C03630=1077.556,71.038,-65.531,173.800,22.783,153.961
C03631=1077.550,70.789,-65.513,173.799,22.780,153.960
C03632=1077.544,70.540,-65.497,173.797,22.778,153.960
C03633=1077.539,70.291,-65.480,173.796,22.775,153.960
C03634=1077.533,70.041,-65.462,173.794,22.773,153.959
C03635=1077.527,69.791,-65.445,173.793,22.770,153.959
C03636=1077.521,69.542,-65.428,173.791,22.768,153.959
C03637=1077.516,69.293,-65.411,173.790,22.765,153.959
C03638=1077.510,69.044,-65.394,173.788,22.763,153.958
C03639=1077.504,68.794,-65.377,173.786,22.760,153.958
C03640=1077.498,68.545,-65.360,173.785,22.758,153.958
C03641=1077.492,68.295,-65.343,173.784,22.756,153.958
C03642=1077.486,68.046,-65.327,173.782,22.753,153.957
C03643=1077.481,67.797,-65.309,173.780,22.750,153.957
C03644=1077.475,67.548,-65.293,173.779,22.748,153.957
C03645=1077.469,67.298,-65.275,173.778,22.746,153.957
C03646=1077.464,67.048,-65.258,173.775,22.743,153.956
C03647=1077.457,66.799,-65.241,173.774,22.741,153.956
C03648=1077.452,66.550,-65.224,173.773,22.738,153.956
C03649=1077.446,66.300,-65.208,173.771,22.736,153.955
C03650=1077.441,66.051,-65.191,173.770,22.733,153.955
C03651=1077.435,65.802,-65.174,173.768,22.731,153.955
C03652=1077.429,65.552,-65.156,173.767,22.729,153.955
C03653=1077.423,65.303,-65.140,173.765,22.726,153.954
C03654=1077.417,65.053,-65.123,173.763,22.724,153.954
C03655=1077.411,64.804,-65.106,173.762,22.721,153.954
C03656=1077.406,64.555,-65.089,173.760,22.718,153.954
C03657=1077.400,64.305,-65.073,173.759,22.716,153.953
C03658=1077.394,64.057,-65.056,173.758,22.713,153.953
C03659=1077.389,63.807,-65.039,173.756,22.712,153.953
C03660=1077.382,63.557,-65.023,173.754,22.709,153.953
C03661=1077.376,63.277,-65.004,173.753,22.706,153.952
C03662=1077.369,62.996,-64.985,173.751,22.703,153.952
C03663=1077.362,62.715,-64.966,173.750,22.701,153.952
C03664=1077.356,62.435,-64.947,173.747,22.698,153.951
C03665=1077.349,62.185,-64.930,173.746,22.695,153.951
C03666=1077.343,61.936,-64.914,173.745,22.693,153.951
C03667=1077.338,61.686,-64.898,173.743,22.691,153.951
C03668=1077.332,61.437,-64.880,173.741,22.688,153.950
C03669=1077.326,61.188,-64.864,173.740,22.686,153.950
C03670=1077.320,60.938,-64.848,173.738,22.683,153.950
C03671=1077.314,60.689,-64.832,173.737,22.680,153.950
C03672=1077.309,60.439,-64.815,173.735,22.679,153.949
C03673=1077.303,60.191,-64.798,173.734,22.676,153.949
C03674=1077.296,59.941,-64.781,173.732,22.673,153.949
C03675=1077.291,59.691,-64.764,173.731,22.671,153.949
C03676=1077.285,59.442,-64.748,173.730,22.668,153.948
C03677=1077.279,59.192,-64.732,173.728,22.666,153.948
C03678=1077.273,58.943,-64.716,173.726,22.664,153.948
C03679=1077.268,58.694,-64.698,173.725,22.661,153.948
C03680=1077.262,58.445,-64.682,173.724,22.659,153.947
C03681=1077.256,58.195,-64.665,173.721,22.656,153.947
C03682=1077.250,57.946,-64.649,173.720,22.654,153.947
C03683=1077.244,57.696,-64.632,173.719,22.651,153.946
C03684=1077.239,57.447,-64.616,173.718,22.649,153.946
C03685=1077.233,57.198,-64.600,173.715,22.646,153.946
C03686=1077.227,56.948,-64.584,173.714,22.644,153.946
C03687=1077.221,56.699,-64.567,173.713,22.642,153.945
C03688=1077.215,56.450,-64.550,173.712,22.639,153.945
C03689=1077.209,56.200,-64.534,173.710,22.636,153.945
C03690=1077.203,55.951,-64.517,173.708,22.634,153.945
C03691=1077.197,55.702,-64.501,173.707,22.631,153.944
C03692=1077.191,55.452,-64.485,173.706,22.629,153.944
C03693=1077.186,55.203,-64.468,173.704,22.626,153.944
C03694=1077.180,54.953,-64.452,173.702,22.624,153.944
C03695=1077.174,54.704,-64.435,173.701,22.622,153.943
C03696=1077.168,54.455,-64.419,173.700,22.619,153.943
C03697=1077.162,54.205,-64.403,173.698,22.617,153.943
C03698=1077.157,53.956,-64.386,173.696,22.614,153.942
C03699=1077.151,53.706,-64.370,173.695,22.612,153.942
C03700=1077.145,53.457,-64.354,173.694,22.609,153.942
C03701=1077.139,53.208,-64.337,173.692,22.606,153.942
C03702=1077.133,52.958,-64.321,173.691,22.604,153.941
C03703=1077.128,52.709,-64.304,173.689,22.602,153.941
C03704=1077.122,52.459,-64.288,173.688,22.599,153.941
C03705=1077.116,52.210,-64.272,173.686,22.596,153.940
C03706=1077.110,51.961,-64.255,173.685,22.594,153.940
C03707=1077.105,51.711,-64.240,173.683,22.592,153.940
C03708=1077.099,51.461,-64.224,173.681,22.589,153.940
C03709=1077.093,51.212,-64.207,173.680,22.587,153.939
C03710=1077.087,50.962,-64.190,173.679,22.584,153.939
C03711=1077.082,50.713,-64.174,173.678,22.582,153.939
C03712=1077.076,50.464,-64.158,173.675,22.579,153.939
C03713=1077.070,50.215,-64.142,173.674,22.577,153.938
C03714=1077.064,49.966,-64.126,173.673,22.574,153.938
C03715=1077.059,49.716,-64.110,173.672,22.572,153.938
C03716=1077.053,49.466,-64.093,173.670,22.569,153.937
C03717=1077.047,49.217,-64.077,173.668,22.566,153.937
C03718=1077.042,48.967,-64.061,173.667,22.564,153.937
C03719=1077.036,48.718,-64.045,173.666,22.562,153.937
C03720=1077.030,48.469,-64.028,173.665,22.559,153.936
C03721=1077.024,48.219,-64.013,173.663,22.556,153.936
C03722=1077.019,47.970,-63.997,173.661,22.554,153.936
C03723=1077.013,47.721,-63.981,173.660,22.551,153.935
C03724=1077.007,47.471,-63.964,173.659,22.549,153.935
C03725=1077.000,47.189,-63.946,173.657,22.546,153.935
C03726=1076.994,46.909,-63.928,173.655,22.543,153.935
C03727=1076.988,46.628,-63.909,173.654,22.540,153.934
C03728=1076.982,46.347,-63.892,173.651,22.538,153.934
C03729=1076.976,46.097,-63.875,173.650,22.535,153.934
C03730=1076.970,45.848,-63.859,173.649,22.533,153.933
C03731=1076.964,45.599,-63.843,173.648,22.530,153.933
C03732=1076.959,45.349,-63.828,173.646,22.527,153.933
C03733=1076.953,45.100,-63.812,173.644,22.525,153.932
C03734=1076.947,44.851,-63.795,173.643,22.523,153.932
C03735=1076.941,44.601,-63.780,173.642,22.520,153.932
C03736=1076.936,44.351,-63.763,173.641,22.518,153.932
C03737=1076.930,44.103,-63.748,173.639,22.515,153.931
C03738=1076.925,43.853,-63.732,173.637,22.512,153.931
C03739=1076.919,43.603,-63.716,173.636,22.510,153.931
C03740=1076.913,43.354,-63.700,173.635,22.508,153.930
C03741=1076.907,43.104,-63.684,173.633,22.505,153.930
C03742=1076.901,42.855,-63.668,173.632,22.502,153.930
C03743=1076.896,42.606,-63.652,173.630,22.500,153.930
C03744=1076.890,42.356,-63.636,173.629,22.497,153.929
C03745=1076.884,42.107,-63.620,173.627,22.494,153.929
C03746=1076.878,41.857,-63.605,173.626,22.492,153.929
C03747=1076.872,41.608,-63.589,173.625,22.490,153.928
C03748=1076.866,41.359,-63.573,173.623,22.488,153.928
C03749=1076.861,41.109,-63.557,173.621,22.485,153.928
C03750=1076.855,40.860,-63.541,173.620,22.482,153.928
C03751=1076.849,40.610,-63.526,173.619,22.480,153.927
C03752=1076.843,40.360,-63.509,173.617,22.478,153.927
C03753=1076.838,40.111,-63.494,173.616,22.475,153.927
C03754=1076.831,39.862,-63.479,173.614,22.472,153.927
C03755=1076.826,39.613,-63.462,173.613,22.470,153.926
C03756=1076.820,39.363,-63.447,173.612,22.467,153.926
C03757=1076.814,39.113,-63.430,173.610,22.465,153.926
C03758=1076.809,38.864,-63.415,173.608,22.462,153.925
C03759=1076.803,38.615,-63.399,173.607,22.460,153.925
C03760=1076.797,38.365,-63.383,173.606,22.457,153.925
C03761=1076.791,38.116,-63.368,173.605,22.455,153.925
C03762=1076.786,37.867,-63.353,173.603,22.452,153.924
C03763=1076.780,37.617,-63.337,173.601,22.449,153.924
C03764=1076.774,37.367,-63.321,173.600,22.448,153.924
C03765=1076.768,37.118,-63.306,173.599,22.445,153.924
C03766=1076.762,36.869,-63.290,173.597,22.443,153.923
C03767=1076.757,36.619,-63.274,173.595,22.440,153.923
C03768=1076.750,36.370,-63.259,173.594,22.437,153.923
C03769=1076.744,36.120,-63.243,173.593,22.435,153.922
C03770=1076.738,35.871,-63.227,173.592,22.433,153.922
C03771=1076.732,35.622,-63.212,173.590,22.430,153.922
C03772=1076.727,35.372,-63.197,173.588,22.427,153.922
C03773=1076.721,35.122,-63.181,173.587,22.425,153.921
C03774=1076.715,34.873,-63.166,173.586,22.423,153.921
C03775=1076.709,34.624,-63.150,173.584,22.420,153.921
C03776=1076.704,34.374,-63.134,173.582,22.418,153.921
C03777=1076.697,34.124,-63.119,173.581,22.415,153.920
C03778=1076.691,33.875,-63.103,173.580,22.413,153.920
C03779=1076.686,33.626,-63.088,173.579,22.410,153.920
C03780=1076.680,33.376,-63.073,173.577,22.408,153.919
C03781=1076.674,33.127,-63.057,173.575,22.405,153.919
C03782=1076.669,32.878,-63.042,173.574,22.403,153.919
C03783=1076.662,32.628,-63.027,173.573,22.400,153.919
C03784=1076.656,32.379,-63.010,173.571,22.398,153.918
C03785=1076.651,32.130,-62.996,173.570,22.396,153.918
C03786=1076.645,31.880,-62.980,173.568,22.393,153.918
C03787=1076.639,31.630,-62.965,173.567,22.390,153.918
C03788=1076.633,31.381,-62.949,173.566,22.388,153.917
C03789=1076.626,31.100,-62.932,173.564,22.385,153.917
C03790=1076.620,30.819,-62.914,173.563,22.382,153.917
C03791=1076.614,30.538,-62.897,173.560,22.379,153.916
C03792=1076.607,30.256,-62.880,173.559,22.377,153.916
C03793=1076.602,30.007,-62.865,173.558,22.374,153.916
C03794=1076.595,29.757,-62.850,173.557,22.372,153.916
C03795=1076.590,29.509,-62.834,173.555,22.369,153.915
C03796=1076.584,29.259,-62.819,173.553,22.367,153.915
C03797=1076.578,29.009,-62.803,173.552,22.364,153.915
C03798=1076.573,28.760,-62.788,173.551,22.362,153.914
C03799=1076.567,28.510,-62.773,173.550,22.359,153.914
C03800=1076.561,28.261,-62.757,173.548,22.356,153.914
C03801=1076.555,28.012,-62.742,173.546,22.354,153.914
C03802=1076.548,27.762,-62.727,173.545,22.352,153.913
C03803=1076.543,27.512,-62.712,173.544,22.350,153.913
C03804=1076.537,27.263,-62.697,173.543,22.347,153.913
C03805=1076.531,27.013,-62.682,173.541,22.344,153.913
C03806=1076.525,26.764,-62.666,173.539,22.342,153.912
C03807=1076.520,26.515,-62.651,173.538,22.339,153.912
C03808=1076.513,26.265,-62.636,173.537,22.337,153.912
C03809=1076.508,26.015,-62.620,173.536,22.335,153.911
C03810=1076.502,25.767,-62.606,173.533,22.332,153.911
C03811=1076.495,25.517,-62.591,173.532,22.330,153.911
C03812=1076.490,25.268,-62.576,173.531,22.327,153.911
C03813=1076.484,25.018,-62.561,173.530,22.325,153.910
C03814=1076.478,24.768,-62.545,173.528,22.322,153.910
C03815=1076.473,24.519,-62.531,173.526,22.320,153.910
C03816=1076.467,24.269,-62.515,173.525,22.317,153.910
C03817=1076.461,24.019,-62.500,173.524,22.315,153.909
C03818=1076.455,23.770,-62.486,173.523,22.313,153.909
C03819=1076.449,23.520,-62.470,173.521,22.310,153.909
C03820=1076.443,23.271,-62.455,173.519,22.307,153.909
C03821=1076.437,23.022,-62.441,173.518,22.305,153.908
C03822=1076.431,22.772,-62.425,173.517,22.303,153.908
C03823=1076.426,22.523,-62.410,173.516,22.300,153.908
C03824=1076.420,22.273,-62.395,173.514,22.298,153.907
C03825=1076.414,22.024,-62.380,173.512,22.295,153.907
C03826=1076.408,21.774,-62.365,173.511,22.293,153.907
C03827=1076.403,21.525,-62.350,173.510,22.290,153.907
C03828=1076.396,21.275,-62.335,173.508,22.288,153.906
C03829=1076.391,21.026,-62.321,173.507,22.286,153.906
C03830=1076.385,20.776,-62.305,173.505,22.283,153.906
C03831=1076.379,20.527,-62.290,173.504,22.280,153.906
C03832=1076.373,20.278,-62.275,173.503,22.278,153.905
C03833=1076.367,20.028,-62.260,173.502,22.275,153.905
C03834=1076.361,19.779,-62.245,173.500,22.273,153.905
C03835=1076.355,19.529,-62.231,173.498,22.271,153.905
C03836=1076.350,19.280,-62.215,173.497,22.268,153.904
C03837=1076.344,19.030,-62.200,173.496,22.266,153.904
C03838=1076.338,18.781,-62.187,173.494,22.263,153.904
C03839=1076.332,18.531,-62.172,173.493,22.261,153.903
C03840=1076.327,18.282,-62.156,173.491,22.258,153.903
C03841=1076.320,18.032,-62.141,173.490,22.256,153.903
C03842=1076.314,17.783,-62.127,173.488,22.254,153.903
C03843=1076.308,17.534,-62.112,173.487,22.251,153.902
C03844=1076.302,17.284,-62.096,173.486,22.249,153.902
C03845=1076.297,17.034,-62.083,173.485,22.246,153.902
C03846=1076.291,16.784,-62.068,173.483,22.243,153.902
C03847=1076.285,16.535,-62.053,173.482,22.241,153.901
C03848=1076.278,16.286,-62.038,173.480,22.239,153.901
C03849=1076.273,16.037,-62.023,173.479,22.236,153.901
C03850=1076.267,15.786,-62.009,173.478,22.234,153.900
C03851=1076.262,15.537,-61.994,173.476,22.231,153.900
C03852=1076.255,15.288,-61.979,173.474,22.229,153.900
C03853=1076.250,15.008,-61.963,173.473,22.226,153.900
C03854=1076.243,14.729,-61.946,173.471,22.223,153.899
C03855=1076.236,14.449,-61.930,173.470,22.220,153.899
C03856=1076.230,14.170,-61.914,173.468,22.218,153.899
C03857=1076.223,13.920,-61.899,173.467,22.216,153.899
C03858=1076.217,13.671,-61.884,173.465,22.213,153.898
C03859=1076.211,13.421,-61.870,173.464,22.211,153.898
C03860=1076.206,13.172,-61.856,173.463,22.208,153.898
C03861=1076.199,12.922,-61.841,173.462,22.206,153.898
C03862=1076.193,12.673,-61.826,173.460,22.203,153.897
C03863=1076.187,12.423,-61.812,173.458,22.201,153.897
C03864=1076.182,12.174,-61.797,173.457,22.199,153.897
C03865=1076.175,11.924,-61.782,173.456,22.196,153.896
C03866=1076.170,11.675,-61.768,173.455,22.194,153.896
C03867=1076.163,11.425,-61.753,173.453,22.192,153.896
C03868=1076.158,11.176,-61.739,173.451,22.189,153.896
C03869=1076.151,10.926,-61.725,173.450,22.186,153.895
C03870=1076.146,10.677,-61.710,173.449,22.184,153.895
C03871=1076.140,10.427,-61.696,173.447,22.182,153.895
C03872=1076.134,10.178,-61.681,173.446,22.180,153.895
C03873=1076.127,9.928,-61.666,173.444,22.177,153.894
C03874=1076.122,9.678,-61.652,173.443,22.175,153.894
C03875=1076.116,9.429,-61.637,173.442,22.172,153.894
C03876=1076.110,9.179,-61.624,173.440,22.170,153.894
C03877=1076.104,8.930,-61.609,173.439,22.167,153.893
C03878=1076.098,8.681,-61.594,173.438,22.165,153.893
C03879=1076.092,8.431,-61.580,173.436,22.163,153.893
C03880=1076.086,8.181,-61.565,173.434,22.160,153.893
C03881=1076.081,7.932,-61.551,173.433,22.158,153.892
C03882=1076.074,7.682,-61.536,173.432,22.155,153.892
C03883=1076.069,7.432,-61.523,173.431,22.153,153.892
C03884=1076.063,7.184,-61.508,173.429,22.151,153.892
C03885=1076.057,6.933,-61.494,173.427,22.148,153.891
C03886=1076.051,6.684,-61.479,173.426,22.146,153.891
C03887=1076.045,6.434,-61.465,173.425,22.143,153.891
C03888=1076.039,6.185,-61.450,173.424,22.141,153.891
C03889=1076.034,5.935,-61.437,173.422,22.139,153.890
C03890=1076.027,5.686,-61.422,173.421,22.136,153.890
C03891=1076.022,5.436,-61.408,173.419,22.133,153.890
C03892=1076.016,5.187,-61.393,173.418,22.131,153.890
C03893=1076.009,4.937,-61.379,173.416,22.129,153.889
C03894=1076.004,4.688,-61.365,173.415,22.127,153.889
C03895=1075.998,4.439,-61.351,173.414,22.124,153.889
C03896=1075.992,4.189,-61.337,173.412,22.121,153.889
C03897=1075.986,3.940,-61.322,173.411,22.119,153.888
C03898=1075.980,3.689,-61.308,173.409,22.117,153.888
C03899=1075.974,3.440,-61.293,173.408,22.114,153.888
C03900=1075.969,3.191,-61.280,173.407,22.112,153.887
C03901=1075.963,2.941,-61.266,173.406,22.109,153.887
C03902=1075.957,2.692,-61.251,173.403,22.107,153.887
C03903=1075.952,2.442,-61.237,173.402,22.105,153.887
C03904=1075.945,2.193,-61.223,173.401,22.102,153.887
C03905=1075.939,1.943,-61.209,173.400,22.100,153.886
C03906=1075.933,1.693,-61.195,173.399,22.098,153.886
C03907=1075.928,1.444,-61.180,173.397,22.095,153.886
C03908=1075.922,1.194,-61.166,173.395,22.092,153.886
C03909=1075.916,0.945,-61.152,173.394,22.090,153.885
C03910=1075.910,0.696,-61.138,173.393,22.088,153.885
C03911=1075.905,0.446,-61.124,173.391,22.086,153.885
C03912=1075.899,0.196,-61.109,173.390,22.083,153.884
C03913=1075.893,-0.053,-61.096,173.389,22.081,153.884
C03914=1075.887,-0.302,-61.082,173.387,22.078,153.884
C03915=1075.881,-0.553,-61.067,173.386,22.075,153.884
C03916=1075.875,-0.802,-61.054,173.384,22.073,153.883
C03917=1075.869,-1.080,-61.038,173.383,22.071,153.883
C03918=1075.862,-1.357,-61.023,173.381,22.068,153.883
C03919=1075.857,-1.635,-61.006,173.380,22.065,153.883
C03920=1075.849,-1.913,-60.991,173.379,22.063,153.882
C03921=1075.844,-2.162,-60.977,173.377,22.060,153.882
C03922=1075.837,-2.411,-60.963,173.375,22.058,153.882
C03923=1075.832,-2.661,-60.949,173.374,22.055,153.882
C03924=1075.826,-2.910,-60.935,173.373,22.053,153.881
C03925=1075.820,-3.161,-60.921,173.372,22.050,153.881
C03926=1075.815,-3.410,-60.907,173.370,22.048,153.881
C03927=1075.808,-3.659,-60.893,173.368,22.046,153.881
C03928=1075.803,-3.908,-60.879,173.367,22.043,153.880
C03929=1075.796,-4.158,-60.865,173.366,22.041,153.880
C03930=1075.791,-4.408,-60.852,173.365,22.039,153.880
C03931=1075.785,-4.657,-60.838,173.363,22.036,153.880
C03932=1075.778,-4.907,-60.823,173.362,22.034,153.879
C03933=1075.773,-5.156,-60.810,173.360,22.031,153.879
C03934=1075.767,-5.406,-60.796,173.359,22.030,153.879
C03935=1075.761,-5.655,-60.782,173.357,22.027,153.879
C03936=1075.755,-5.905,-60.768,173.356,22.025,153.878
C03937=1075.749,-6.155,-60.755,173.355,22.023,153.878
C03938=1075.743,-6.404,-60.741,173.354,22.020,153.878
C03939=1075.737,-6.654,-60.728,173.352,22.018,153.878
C03940=1075.731,-6.904,-60.714,173.350,22.015,153.878
C03941=1075.725,-7.153,-60.699,173.349,22.013,153.877
C03942=1075.719,-7.402,-60.686,173.348,22.010,153.877
C03943=1075.713,-7.652,-60.672,173.346,22.009,153.877
C03944=1075.707,-7.901,-60.659,173.345,22.006,153.876
C03945=1075.701,-8.151,-60.644,173.344,22.004,153.876
C03946=1075.696,-8.401,-60.630,173.342,22.001,153.876
C03947=1075.689,-8.650,-60.617,173.341,21.999,153.876
C03948=1075.684,-8.900,-60.603,173.339,21.997,153.876
C03949=1075.678,-9.149,-60.590,173.338,21.994,153.875
C03950=1075.672,-9.399,-60.576,173.337,21.992,153.875
C03951=1075.665,-9.648,-60.563,173.335,21.990,153.875
C03952=1075.660,-9.898,-60.549,173.334,21.988,153.875
C03953=1075.654,-10.147,-60.535,173.332,21.985,153.874
C03954=1075.648,-10.397,-60.522,173.331,21.983,153.874
C03955=1075.641,-10.647,-60.508,173.330,21.980,153.874
C03956=1075.636,-10.896,-60.494,173.328,21.978,153.874
C03957=1075.630,-11.146,-60.480,173.327,21.976,153.873
C03958=1075.624,-11.395,-60.467,173.326,21.973,153.873
C03959=1075.619,-11.645,-60.453,173.323,21.971,153.873
C03960=1075.613,-11.894,-60.440,173.322,21.969,153.873
C03961=1075.607,-12.144,-60.426,173.321,21.966,153.872
C03962=1075.600,-12.394,-60.412,173.320,21.964,153.872
C03963=1075.595,-12.644,-60.399,173.319,21.962,153.872
C03964=1075.589,-12.893,-60.386,173.317,21.959,153.872
C03965=1075.583,-13.143,-60.372,173.316,21.957,153.872
C03966=1075.577,-13.392,-60.359,173.314,21.954,153.871
C03967=1075.572,-13.641,-60.345,173.313,21.952,153.871
C03968=1075.565,-13.891,-60.332,173.311,21.950,153.871
C03969=1075.560,-14.140,-60.318,173.310,21.948,153.871
C03970=1075.554,-14.390,-60.304,173.309,21.946,153.870
C03971=1075.548,-14.640,-60.291,173.308,21.943,153.870
C03972=1075.542,-14.890,-60.278,173.306,21.941,153.870
C03973=1075.536,-15.139,-60.264,173.304,21.938,153.870
C03974=1075.530,-15.389,-60.251,173.303,21.936,153.869
C03975=1075.524,-15.638,-60.237,173.302,21.934,153.869
C03976=1075.518,-15.887,-60.223,173.300,21.931,153.869
C03977=1075.513,-16.137,-60.211,173.299,21.930,153.869
C03978=1075.506,-16.387,-60.198,173.298,21.927,153.869
C03979=1075.500,-16.637,-60.183,173.296,21.925,153.868
C03980=1075.494,-16.886,-60.170,173.294,21.922,153.868
C03981=1075.488,-17.162,-60.156,173.293,21.920,153.868
C03982=1075.481,-17.437,-60.141,173.292,21.918,153.868
C03983=1075.474,-17.714,-60.126,173.290,21.915,153.867
C03984=1075.468,-17.990,-60.112,173.289,21.912,153.867
C03985=1075.462,-18.240,-60.098,173.287,21.911,153.867
C03986=1075.456,-18.489,-60.085,173.286,21.908,153.867
C03987=1075.450,-18.738,-60.071,173.284,21.906,153.867
C03988=1075.444,-18.988,-60.059,173.283,21.903,153.866
C03989=1075.438,-19.237,-60.045,173.281,21.901,153.866
C03990=1075.432,-19.487,-60.032,173.280,21.899,153.866
C03991=1075.426,-19.736,-60.018,173.279,21.897,153.866
C03992=1075.420,-19.986,-60.006,173.277,21.894,153.865
C03993=1075.413,-20.236,-59.992,173.276,21.892,153.865
C03994=1075.408,-20.486,-59.978,173.275,21.890,153.865
C03995=1075.402,-20.736,-59.966,173.273,21.888,153.865
C03996=1075.396,-20.985,-59.952,173.271,21.885,153.865
C03997=1075.390,-21.234,-59.939,173.270,21.883,153.864
C03998=1075.384,-21.484,-59.926,173.269,21.881,153.864
C03999=1075.378,-21.734,-59.913,173.267,21.879,153.864
C04000=1075.372,-21.983,-59.900,173.266,21.876,153.864
C04001=1075.367,-22.233,-59.886,173.265,21.874,153.863
C04002=1075.361,-22.482,-59.873,173.263,21.872,153.863
C04003=1075.355,-22.732,-59.861,173.261,21.870,153.863
C04004=1075.348,-22.981,-59.847,173.260,21.867,153.863
C04005=1075.343,-23.231,-59.833,173.259,21.865,153.863
C04006=1075.337,-23.481,-59.821,173.258,21.863,153.862
C04007=1075.331,-23.730,-59.808,173.256,21.861,153.862
C04008=1075.325,-23.980,-59.795,173.255,21.858,153.862
C04009=1075.319,-24.229,-59.782,173.253,21.856,153.862
C04010=1075.313,-24.479,-59.768,173.252,21.853,153.861
C04011=1075.307,-24.729,-59.755,173.250,21.852,153.861
C04012=1075.301,-24.978,-59.742,173.249,21.849,153.861
C04013=1075.295,-25.228,-59.730,173.248,21.847,153.861
C04014=1075.290,-25.478,-59.716,173.246,21.845,153.861
C04015=1075.284,-25.727,-59.703,173.245,21.843,153.860
C04016=1075.278,-25.977,-59.690,173.244,21.841,153.860
C04017=1075.272,-26.227,-59.677,173.242,21.838,153.860
C04018=1075.266,-26.475,-59.664,173.240,21.836,153.860
C04019=1075.261,-26.725,-59.651,173.239,21.833,153.860
C04020=1075.255,-26.975,-59.638,173.238,21.832,153.859
C04021=1075.249,-27.224,-59.625,173.237,21.829,153.859
C04022=1075.243,-27.474,-59.612,173.235,21.827,153.859
C04023=1075.237,-27.724,-59.600,173.234,21.825,153.859
C04024=1075.230,-27.973,-59.586,173.232,21.822,153.859
C04025=1075.225,-28.223,-59.574,173.230,21.820,153.858
C04026=1075.218,-28.472,-59.560,173.229,21.818,153.858
C04027=1075.212,-28.722,-59.548,173.228,21.816,153.858
C04028=1075.207,-28.972,-59.535,173.227,21.814,153.858
C04029=1075.200,-29.221,-59.522,173.225,21.812,153.858
C04030=1075.194,-29.471,-59.510,173.224,21.810,153.857
C04031=1075.188,-29.720,-59.496,173.223,21.808,153.857
C04032=1075.182,-29.970,-59.484,173.220,21.805,153.857
C04033=1075.176,-30.220,-59.471,173.219,21.803,153.857
C04034=1075.170,-30.469,-59.458,173.218,21.801,153.857
C04035=1075.164,-30.719,-59.445,173.216,21.799,153.856
C04036=1075.158,-30.968,-59.432,173.215,21.796,153.856
C04037=1075.152,-31.218,-59.420,173.214,21.795,153.856
C04038=1075.146,-31.468,-59.407,173.212,21.793,153.856
C04039=1075.140,-31.717,-59.394,173.211,21.790,153.856
C04040=1075.134,-31.967,-59.381,173.209,21.788,153.855
C04041=1075.129,-32.216,-59.369,173.208,21.786,153.855
C04042=1075.123,-32.466,-59.356,173.207,21.783,153.855
C04043=1075.117,-32.716,-59.343,173.205,21.781,153.855
C04044=1075.111,-32.966,-59.331,173.204,21.779,153.855
C04045=1075.104,-33.240,-59.316,173.203,21.777,153.854
C04046=1075.097,-33.516,-59.303,173.200,21.775,153.854
C04047=1075.091,-33.791,-59.289,173.199,21.772,153.854
C04048=1075.084,-34.066,-59.274,173.198,21.770,153.854
C04049=1075.078,-34.316,-59.262,173.197,21.768,153.854
C04050=1075.072,-34.566,-59.249,173.194,21.765,153.853
C04051=1075.066,-34.814,-59.236,173.193,21.763,153.853
C04052=1075.061,-35.064,-59.224,173.192,21.761,153.853
C04053=1075.055,-35.314,-59.211,173.190,21.759,153.853
C04054=1075.049,-35.564,-59.199,173.189,21.757,153.853
C04055=1075.043,-35.814,-59.186,173.188,21.755,153.852
C04056=1075.037,-36.063,-59.173,173.187,21.753,153.852
C04057=1075.031,-36.313,-59.160,173.185,21.751,153.852
C04058=1075.025,-36.562,-59.149,173.183,21.748,153.852
C04059=1075.019,-36.812,-59.136,173.182,21.746,153.852
C04060=1075.013,-37.062,-59.124,173.180,21.744,153.852
C04061=1075.007,-37.311,-59.110,173.179,21.742,153.851
C04062=1075.001,-37.561,-59.098,173.178,21.740,153.851
C04063=1074.995,-37.810,-59.086,173.176,21.738,153.851
C04064=1074.989,-38.060,-59.073,173.175,21.736,153.851
C04065=1074.984,-38.310,-59.060,173.174,21.734,153.851
C04066=1074.978,-38.560,-59.048,173.173,21.731,153.850
C04067=1074.971,-38.809,-59.035,173.170,21.729,153.850
C04068=1074.965,-39.058,-59.023,173.169,21.727,153.850
C04069=1074.959,-39.308,-59.011,173.168,21.725,153.850
C04070=1074.954,-39.557,-58.998,173.166,21.723,153.850
C04071=1074.947,-39.807,-58.986,173.165,21.721,153.850
C04072=1074.941,-40.057,-58.973,173.164,21.719,153.849
C04073=1074.935,-40.307,-58.961,173.162,21.717,153.849
C04074=1074.929,-40.557,-58.948,173.161,21.715,153.849
C04075=1074.923,-40.806,-58.937,173.159,21.713,153.849
C04076=1074.917,-41.055,-58.923,173.157,21.710,153.849
C04077=1074.911,-41.305,-58.911,173.156,21.708,153.849
C04078=1074.905,-41.555,-58.898,173.154,21.707,153.848
C04079=1074.898,-41.804,-58.886,173.153,21.704,153.848
C04080=1074.893,-42.053,-58.874,173.152,21.702,153.848
C04081=1074.887,-42.303,-58.862,173.151,21.700,153.848
C04082=1074.881,-42.553,-58.850,173.149,21.698,153.848
C04083=1074.875,-42.803,-58.837,173.148,21.696,153.848
C04084=1074.869,-43.053,-58.825,173.146,21.694,153.847
C04085=1074.863,-43.301,-58.813,173.144,21.692,153.847
C04086=1074.857,-43.551,-58.800,173.143,21.690,153.847
C04087=1074.851,-43.801,-58.788,173.142,21.688,153.847
C04088=1074.844,-44.051,-58.776,173.140,21.686,153.847
C04089=1074.839,-44.300,-58.764,173.139,21.684,153.846
C04090=1074.833,-44.550,-58.751,173.138,21.682,153.846
C04091=1074.827,-44.800,-58.739,173.136,21.680,153.846
C04092=1074.821,-45.049,-58.727,173.135,21.678,153.846
C04093=1074.815,-45.298,-58.715,173.133,21.676,153.846
C04094=1074.809,-45.548,-58.702,173.132,21.674,153.846
C04095=1074.803,-45.798,-58.690,173.130,21.672,153.846
C04096=1074.797,-46.048,-58.678,173.129,21.669,153.845
C04097=1074.791,-46.297,-58.667,173.127,21.667,153.845
C04098=1074.785,-46.547,-58.654,173.126,21.665,153.845
C04099=1074.779,-46.797,-58.641,173.125,21.663,153.845
C04100=1074.773,-47.046,-58.630,173.123,21.661,153.845
C04101=1074.767,-47.296,-58.617,173.122,21.659,153.845
C04102=1074.761,-47.546,-58.605,173.120,21.657,153.844
C04103=1074.755,-47.795,-58.593,173.119,21.656,153.844
C04104=1074.749,-48.044,-58.581,173.118,21.654,153.844
C04105=1074.743,-48.294,-58.568,173.116,21.651,153.844
C04106=1074.737,-48.545,-58.557,173.114,21.649,153.844
C04107=1074.732,-48.794,-58.545,173.113,21.647,153.844
C04108=1074.726,-49.044,-58.532,173.111,21.645,153.843
C04109=1074.719,-49.319,-58.519,173.110,21.643,153.843
C04110=1074.713,-49.595,-58.506,173.109,21.641,153.843
C04111=1074.706,-49.870,-58.492,173.107,21.639,153.843
C04112=1074.699,-50.146,-58.479,173.105,21.637,153.843
C04113=1074.694,-50.395,-58.467,173.104,21.634,153.842
C04114=1074.688,-50.645,-58.455,173.103,21.633,153.842
C04115=1074.681,-50.895,-58.443,173.101,21.631,153.842
C04116=1074.675,-51.144,-58.431,173.100,21.629,153.842
C04117=1074.669,-51.393,-58.419,173.098,21.626,153.842
C04118=1074.663,-51.644,-58.408,173.096,21.625,153.842
C04119=1074.657,-51.893,-58.395,173.095,21.623,153.842
C04120=1074.650,-52.143,-58.383,173.093,21.621,153.842
C04121=1074.644,-52.392,-58.372,173.092,21.619,153.841
C04122=1074.638,-52.642,-58.360,173.091,21.617,153.841
C04123=1074.632,-52.892,-58.348,173.089,21.615,153.841
C04124=1074.626,-53.141,-58.336,173.088,21.613,153.841
C04125=1074.620,-53.391,-58.324,173.086,21.611,153.841
C04126=1074.613,-53.641,-58.313,173.085,21.610,153.841
C04127=1074.607,-53.890,-58.301,173.084,21.608,153.841
C04128=1074.601,-54.140,-58.288,173.082,21.606,153.840
C04129=1074.595,-54.390,-58.277,173.080,21.604,153.840
C04130=1074.589,-54.639,-58.266,173.079,21.602,153.840
C04131=1074.583,-54.889,-58.253,173.077,21.600,153.840
C04132=1074.577,-55.139,-58.242,173.076,21.598,153.840
C04133=1074.571,-55.388,-58.230,173.074,21.596,153.840
C04134=1074.565,-55.638,-58.218,173.073,21.594,153.840
C04135=1074.559,-55.888,-58.206,173.072,21.593,153.840
C04136=1074.553,-56.137,-58.195,173.070,21.591,153.840
C04137=1074.547,-56.386,-58.182,173.069,21.589,153.839
C04138=1074.540,-56.637,-58.171,173.067,21.587,153.839
C04139=1074.534,-56.886,-58.159,173.066,21.585,153.839
C04140=1074.529,-57.136,-58.148,173.065,21.583,153.839
C04141=1074.522,-57.386,-58.136,173.062,21.581,153.839
C04142=1074.516,-57.634,-58.124,173.061,21.579,153.839
C04143=1074.510,-57.885,-58.113,173.060,21.577,153.839
C04144=1074.504,-58.134,-58.101,173.058,21.575,153.838
C04145=1074.498,-58.384,-58.089,173.057,21.573,153.838
C04146=1074.491,-58.634,-58.077,173.055,21.572,153.838
C04147=1074.486,-58.883,-58.066,173.054,21.570,153.838
C04148=1074.480,-59.133,-58.054,173.053,21.568,153.838
C04149=1074.474,-59.382,-58.042,173.051,21.566,153.838
C04150=1074.467,-59.632,-58.031,173.050,21.564,153.838
C04151=1074.461,-59.882,-58.019,173.048,21.563,153.838
C04152=1074.456,-60.131,-58.008,173.047,21.561,153.837
C04153=1074.449,-60.381,-57.996,173.046,21.559,153.837
C04154=1074.444,-60.631,-57.984,173.044,21.557,153.837
C04155=1074.437,-60.880,-57.972,173.042,21.555,153.837
C04156=1074.432,-61.130,-57.961,173.040,21.553,153.837
C04157=1074.425,-61.379,-57.949,173.039,21.551,153.837
C04158=1074.419,-61.630,-57.938,173.038,21.549,153.837
C04159=1074.413,-61.879,-57.926,173.036,21.548,153.837
C04160=1074.407,-62.129,-57.915,173.035,21.546,153.837
C04161=1074.401,-62.378,-57.903,173.033,21.544,153.836
C04162=1074.395,-62.628,-57.892,173.032,21.542,153.836
C04163=1074.390,-62.878,-57.880,173.030,21.541,153.836
C04164=1074.383,-63.127,-57.868,173.029,21.539,153.836
C04165=1074.377,-63.377,-57.858,173.028,21.537,153.836
C04166=1074.371,-63.626,-57.846,173.026,21.535,153.836
C04167=1074.366,-63.876,-57.834,173.025,21.533,153.836
C04168=1074.359,-64.126,-57.822,173.023,21.531,153.836
C04169=1074.353,-64.375,-57.811,173.022,21.529,153.835
C04170=1074.347,-64.626,-57.800,173.020,21.528,153.835
C04171=1074.341,-64.874,-57.788,173.018,21.526,153.835
C04172=1074.335,-65.125,-57.777,173.017,21.524,153.835
C04173=1074.329,-65.402,-57.765,173.016,21.522,153.835
C04174=1074.322,-65.678,-57.751,173.014,21.520,153.835
C04175=1074.315,-65.956,-57.739,173.012,21.518,153.835
C04176=1074.308,-66.232,-57.726,173.010,21.516,153.835
C04177=1074.302,-66.482,-57.715,173.009,21.514,153.835
C04178=1074.297,-66.731,-57.704,173.008,21.512,153.834
C04179=1074.290,-66.981,-57.692,173.006,21.511,153.834
C04180=1074.285,-67.231,-57.680,173.005,21.509,153.834
C04181=1074.279,-67.481,-57.669,173.003,21.507,153.834
C04182=1074.273,-67.730,-57.658,173.002,21.505,153.834
C04183=1074.266,-67.980,-57.646,173.000,21.503,153.834
C04184=1074.261,-68.229,-57.635,172.999,21.502,153.834
C04185=1074.255,-68.480,-57.624,172.998,21.500,153.834
C04186=1074.249,-68.729,-57.612,172.996,21.498,153.834
C04187=1074.243,-68.978,-57.601,172.995,21.496,153.833
C04188=1074.237,-69.228,-57.590,172.993,21.495,153.833
C04189=1074.231,-69.478,-57.579,172.991,21.492,153.833
C04190=1074.224,-69.727,-57.567,172.990,21.490,153.833
C04191=1074.219,-69.977,-57.556,172.988,21.489,153.833
C04192=1074.214,-70.227,-57.545,172.987,21.487,153.833
C04193=1074.207,-70.477,-57.534,172.985,21.486,153.833
C04194=1074.201,-70.726,-57.522,172.984,21.484,153.833
C04195=1074.195,-70.976,-57.511,172.982,21.482,153.833
C04196=1074.189,-71.225,-57.500,172.981,21.480,153.833
C04197=1074.183,-71.475,-57.489,172.980,21.478,153.832
C04198=1074.177,-71.725,-57.478,172.978,21.477,153.832
C04199=1074.172,-71.974,-57.465,172.977,21.475,153.832
C04200=1074.166,-72.224,-57.455,172.975,21.473,153.832
C04201=1074.160,-72.474,-57.443,172.974,21.472,153.832
C04202=1074.154,-72.723,-57.432,172.972,21.470,153.832
C04203=1074.148,-72.973,-57.422,172.971,21.468,153.832
C04204=1074.142,-73.223,-57.410,172.969,21.466,153.832
C04205=1074.136,-73.472,-57.399,172.968,21.464,153.832
C04206=1074.130,-73.722,-57.388,172.966,21.463,153.832
C04207=1074.125,-73.972,-57.376,172.965,21.461,153.831
C04208=1074.118,-74.221,-57.366,172.964,21.460,153.831
C04209=1074.112,-74.471,-57.355,172.962,21.458,153.831
C04210=1074.106,-74.721,-57.344,172.961,21.456,153.831
C04211=1074.100,-74.970,-57.333,172.959,21.455,153.831
C04212=1074.094,-75.221,-57.322,172.957,21.453,153.831
C04213=1074.088,-75.470,-57.311,172.955,21.451,153.831
C04214=1074.082,-75.720,-57.299,172.954,21.449,153.831
C04215=1074.076,-75.969,-57.288,172.952,21.448,153.831
C04216=1074.070,-76.219,-57.277,172.951,21.446,153.831
C04217=1074.064,-76.469,-57.266,172.949,21.444,153.831
C04218=1074.058,-76.718,-57.255,172.948,21.443,153.831
C04219=1074.052,-76.968,-57.244,172.947,21.441,153.831
C04220=1074.045,-77.218,-57.233,172.945,21.440,153.831
C04221=1074.039,-77.467,-57.222,172.944,21.438,153.830
C04222=1074.034,-77.717,-57.212,172.942,21.436,153.830
C04223=1074.027,-77.967,-57.200,172.941,21.435,153.830
C04224=1074.022,-78.216,-57.189,172.939,21.433,153.830
C04225=1074.016,-78.466,-57.179,172.938,21.432,153.830
C04226=1074.010,-78.716,-57.167,172.936,21.430,153.830
C04227=1074.004,-78.965,-57.156,172.935,21.428,153.830
C04228=1073.998,-79.215,-57.146,172.933,21.427,153.830
C04229=1073.991,-79.465,-57.135,172.932,21.425,153.830
C04230=1073.985,-79.714,-57.124,172.930,21.423,153.830
C04231=1073.979,-79.964,-57.113,172.929,21.422,153.830
C04232=1073.973,-80.214,-57.102,172.927,21.420,153.830
C04233=1073.967,-80.463,-57.092,172.926,21.419,153.830
C04234=1073.961,-80.713,-57.081,172.924,21.417,153.830
C04235=1073.955,-80.963,-57.069,172.923,21.416,153.830
C04236=1073.949,-81.213,-57.059,172.921,21.414,153.829
C04237=1073.942,-81.492,-57.047,172.920,21.412,153.829
C04238=1073.935,-81.770,-57.035,172.917,21.411,153.829
C04239=1073.928,-82.050,-57.023,172.916,21.409,153.829
C04240=1073.921,-82.329,-57.011,172.914,21.407,153.829
C04241=1073.915,-82.578,-57.000,172.913,21.406,153.829
C04242=1073.909,-82.828,-56.989,172.911,21.404,153.829
C04243=1073.902,-83.078,-56.979,172.910,21.403,153.829
C04244=1073.897,-83.328,-56.969,172.908,21.401,153.829
C04245=1073.891,-83.577,-56.958,172.907,21.400,153.829
C04246=1073.884,-83.827,-56.947,172.905,21.398,153.829
C04247=1073.878,-84.077,-56.936,172.904,21.397,153.829
C04248=1073.872,-84.326,-56.925,172.902,21.395,153.829
C04249=1073.865,-84.576,-56.915,172.901,21.394,153.829
C04250=1073.860,-84.826,-56.904,172.899,21.392,153.829
C04251=1073.854,-85.076,-56.894,172.898,21.391,153.829
C04252=1073.848,-85.325,-56.883,172.896,21.389,153.829
C04253=1073.841,-85.575,-56.872,172.895,21.388,153.829
C04254=1073.835,-85.824,-56.862,172.893,21.387,153.829
C04255=1073.829,-86.074,-56.852,172.892,21.385,153.829
C04256=1073.823,-86.325,-56.840,172.890,21.383,153.829
C04257=1073.817,-86.574,-56.830,172.888,21.382,153.829
C04258=1073.811,-86.823,-56.819,172.887,21.380,153.829
C04259=1073.805,-87.073,-56.808,172.885,21.379,153.829
C04260=1073.798,-87.323,-56.798,172.884,21.378,153.829
C04261=1073.793,-87.573,-56.788,172.882,21.376,153.829
C04262=1073.786,-87.822,-56.777,172.881,21.374,153.828
C04263=1073.780,-88.071,-56.766,172.879,21.373,153.828
C04264=1073.775,-88.322,-56.756,172.878,21.371,153.828
C04265=1073.768,-88.571,-56.746,172.876,21.370,153.828
C04266=1073.762,-88.821,-56.735,172.875,21.369,153.828
C04267=1073.757,-89.071,-56.725,172.873,21.367,153.828
C04268=1073.750,-89.320,-56.714,172.872,21.366,153.828
C04269=1073.744,-89.570,-56.703,172.870,21.364,153.828
C04270=1073.737,-89.820,-56.693,172.868,21.363,153.828
C04271=1073.732,-90.070,-56.683,172.867,21.361,153.828
C04272=1073.726,-90.319,-56.672,172.865,21.360,153.828
C04273=1073.720,-90.568,-56.661,172.864,21.359,153.828
C04274=1073.714,-90.819,-56.651,172.862,21.357,153.828
C04275=1073.707,-91.068,-56.641,172.861,21.355,153.828
C04276=1073.702,-91.318,-56.630,172.859,21.354,153.828
C04277=1073.695,-91.568,-56.620,172.858,21.352,153.828
C04278=1073.690,-91.817,-56.609,172.856,21.351,153.828
C04279=1073.684,-92.067,-56.599,172.855,21.350,153.828
C04280=1073.677,-92.317,-56.588,172.853,21.348,153.828
C04281=1073.671,-92.567,-56.578,172.852,21.347,153.828
C04282=1073.665,-92.816,-56.568,172.850,21.345,153.828
C04283=1073.659,-93.066,-56.557,172.848,21.344,153.828
C04284=1073.653,-93.316,-56.548,172.847,21.343,153.828
C04285=1073.648,-93.565,-56.537,172.845,21.341,153.828
C04286=1073.642,-93.815,-56.526,172.844,21.340,153.828
C04287=1073.635,-94.065,-56.516,172.842,21.338,153.828
C04288=1073.629,-94.315,-56.505,172.841,21.337,153.828
C04289=1073.623,-94.564,-56.495,172.839,21.336,153.828
C04290=1073.617,-94.814,-56.485,172.838,21.334,153.828
C04291=1073.611,-95.064,-56.475,172.836,21.333,153.828
C04292=1073.605,-95.313,-56.464,172.834,21.331,153.828
C04293=1073.599,-95.563,-56.455,172.833,21.330,153.828
C04294=1073.594,-95.813,-56.444,172.831,21.329,153.828
C04295=1073.587,-96.062,-56.434,172.830,21.327,153.828
C04296=1073.581,-96.312,-56.423,172.828,21.326,153.828
C04297=1073.575,-96.562,-56.413,172.826,21.325,153.828
C04298=1073.569,-96.812,-56.402,172.825,21.323,153.828
C04299=1073.563,-97.062,-56.393,172.823,21.322,153.828
C04300=1073.557,-97.311,-56.382,172.822,21.321,153.828
C04301=1073.551,-97.592,-56.370,172.820,21.319,153.828
C04302=1073.544,-97.874,-56.360,172.819,21.318,153.828
C04303=1073.537,-98.156,-56.348,172.817,21.316,153.828
C04304=1073.530,-98.436,-56.336,172.815,21.315,153.828
C04305=1073.524,-98.686,-56.326,172.813,21.313,153.828
C04306=1073.518,-98.936,-56.316,172.812,21.312,153.828
C04307=1073.512,-99.185,-56.306,172.810,21.311,153.828
C04308=1073.505,-99.436,-56.295,172.809,21.310,153.828
C04309=1073.499,-99.685,-56.286,172.808,21.308,153.828
C04310=1073.493,-99.934,-56.275,172.806,21.307,153.828
C04311=1073.486,-100.184,-56.266,172.804,21.306,153.828
C04312=1073.481,-100.434,-56.256,172.803,21.305,153.828
C04313=1073.475,-100.684,-56.245,172.801,21.303,153.828
C04314=1073.468,-100.933,-56.236,172.800,21.302,153.828
C04315=1073.463,-101.183,-56.226,172.798,21.301,153.828
C04316=1073.456,-101.433,-56.215,172.796,21.300,153.828
C04317=1073.450,-101.682,-56.206,172.795,21.298,153.828
C04318=1073.445,-101.932,-56.195,172.793,21.297,153.828
C04319=1073.438,-102.182,-56.185,172.792,21.295,153.828
C04320=1073.432,-102.432,-56.175,172.790,21.295,153.828
C04321=1073.426,-102.682,-56.164,172.788,21.293,153.828
C04322=1073.420,-102.932,-56.155,172.787,21.292,153.828
C04323=1073.414,-103.181,-56.145,172.785,21.291,153.828
C04324=1073.407,-103.431,-56.135,172.783,21.290,153.828
C04325=1073.402,-103.681,-56.125,172.782,21.288,153.828
C04326=1073.395,-103.930,-56.115,172.780,21.287,153.828
C04327=1073.389,-104.180,-56.106,172.779,21.286,153.828
C04328=1073.383,-104.429,-56.096,172.777,21.284,153.828
C04329=1073.377,-104.680,-56.085,172.775,21.283,153.828
C04330=1073.371,-104.929,-56.076,172.775,21.283,153.828
C04331=1073.365,-105.178,-56.065,172.773,21.281,153.828
C04332=1073.359,-105.428,-56.056,172.771,21.280,153.828
C04333=1073.353,-105.678,-56.046,172.770,21.279,153.828
C04334=1073.347,-105.928,-56.036,172.768,21.278,153.828
C04335=1073.340,-106.177,-56.026,172.766,21.277,153.828
C04336=1073.334,-106.427,-56.016,172.765,21.275,153.828
C04337=1073.329,-106.677,-56.006,172.763,21.274,153.828
C04338=1073.323,-106.927,-55.997,172.762,21.273,153.828
C04339=1073.317,-107.177,-55.987,172.760,21.272,153.828
C04340=1073.310,-107.426,-55.977,172.758,21.271,153.828
C04341=1073.304,-107.676,-55.967,172.757,21.269,153.828
C04342=1073.298,-107.926,-55.958,172.755,21.268,153.828
C04343=1073.292,-108.176,-55.947,172.753,21.267,153.828
C04344=1073.286,-108.426,-55.938,172.752,21.266,153.828
C04345=1073.280,-108.675,-55.928,172.750,21.265,153.829
C04346=1073.273,-108.925,-55.918,172.749,21.264,153.828
C04347=1073.267,-109.174,-55.908,172.748,21.263,153.829
C04348=1073.261,-109.424,-55.899,172.746,21.262,153.829
C04349=1073.255,-109.674,-55.889,172.744,21.261,153.829
C04350=1073.249,-109.924,-55.880,172.743,21.259,153.829
C04351=1073.242,-110.173,-55.870,172.741,21.258,153.829
C04352=1073.236,-110.423,-55.860,172.739,21.257,153.829
C04353=1073.231,-110.673,-55.850,172.738,21.256,153.829
C04354=1073.225,-110.923,-55.840,172.736,21.255,153.829
C04355=1073.218,-111.172,-55.831,172.734,21.254,153.829
C04356=1073.212,-111.422,-55.821,172.733,21.252,153.829
C04357=1073.206,-111.672,-55.812,172.731,21.252,153.829
C04358=1073.200,-111.922,-55.802,172.729,21.250,153.829
C04359=1073.194,-112.172,-55.792,172.729,21.250,153.829
C04360=1073.187,-112.421,-55.783,172.727,21.249,153.829
C04361=1073.181,-112.671,-55.773,172.725,21.247,153.829
C04362=1073.175,-112.920,-55.763,172.723,21.247,153.829
C04363=1073.169,-113.170,-55.753,172.722,21.245,153.829
C04364=1073.163,-113.419,-55.744,172.720,21.244,153.829
C04365=1073.157,-113.699,-55.733,172.719,21.243,153.829
C04366=1073.150,-113.977,-55.723,172.717,21.242,153.830
C04367=1073.142,-114.256,-55.712,172.715,21.241,153.830
C04368=1073.136,-114.535,-55.701,172.713,21.239,153.830
C04369=1073.130,-114.785,-55.692,172.712,21.239,153.830
C04370=1073.124,-115.035,-55.682,172.710,21.238,153.830
C04371=1073.118,-115.284,-55.672,172.708,21.237,153.830
C04372=1073.112,-115.534,-55.663,172.707,21.236,153.830
C04373=1073.105,-115.784,-55.653,172.705,21.234,153.830
C04374=1073.099,-116.034,-55.644,172.703,21.234,153.830
C04375=1073.093,-116.284,-55.634,172.702,21.233,153.830
C04376=1073.087,-116.533,-55.625,172.700,21.231,153.830
C04377=1073.081,-116.782,-55.616,172.698,21.230,153.830
C04378=1073.074,-117.032,-55.606,172.697,21.230,153.830
C04379=1073.068,-117.282,-55.597,172.695,21.229,153.831
C04380=1073.062,-117.532,-55.587,172.694,21.228,153.830
C04381=1073.056,-117.782,-55.578,172.692,21.227,153.831
C04382=1073.050,-118.032,-55.569,172.691,21.226,153.831
C04383=1073.044,-118.282,-55.559,172.689,21.225,153.831
C04384=1073.038,-118.531,-55.550,172.687,21.224,153.831
C04385=1073.031,-118.781,-55.540,172.686,21.223,153.831
C04386=1073.026,-119.030,-55.531,172.684,21.222,153.831
C04387=1073.020,-119.280,-55.521,172.682,21.221,153.831
C04388=1073.014,-119.530,-55.512,172.680,21.220,153.831
C04389=1073.007,-119.779,-55.503,172.680,21.219,153.831
C04390=1073.000,-120.029,-55.493,172.678,21.218,153.831
C04391=1072.995,-120.280,-55.484,172.676,21.218,153.831
C04392=1072.988,-120.529,-55.475,172.675,21.216,153.831
C04393=1072.982,-120.779,-55.465,172.673,21.215,153.832
C04394=1072.977,-121.028,-55.456,172.671,21.214,153.832
C04395=1072.971,-121.278,-55.447,172.669,21.214,153.832
C04396=1072.964,-121.528,-55.437,172.667,21.213,153.832
C04397=1072.958,-121.778,-55.429,172.666,21.212,153.832
C04398=1072.952,-122.028,-55.419,172.665,21.211,153.832
C04399=1072.945,-122.278,-55.410,172.663,21.210,153.832
C04400=1072.940,-122.527,-55.400,172.662,21.209,153.832
C04401=1072.934,-122.776,-55.391,172.660,21.208,153.832
C04402=1072.927,-123.026,-55.381,172.658,21.207,153.832
C04403=1072.921,-123.276,-55.373,172.656,21.207,153.833
C04404=1072.915,-123.526,-55.363,172.654,21.206,153.833
C04405=1072.909,-123.776,-55.354,172.653,21.204,153.833
C04406=1072.903,-124.025,-55.345,172.652,21.204,153.833
C04407=1072.897,-124.275,-55.336,172.650,21.203,153.833
C04408=1072.891,-124.525,-55.326,172.649,21.202,153.833
C04409=1072.884,-124.775,-55.317,172.647,21.201,153.833
C04410=1072.878,-125.024,-55.308,172.645,21.200,153.833
C04411=1072.873,-125.274,-55.299,172.643,21.200,153.833
C04412=1072.866,-125.524,-55.290,172.641,21.199,153.833
C04413=1072.859,-125.773,-55.281,172.640,21.198,153.834
C04414=1072.853,-126.023,-55.271,172.639,21.197,153.834
C04415=1072.847,-126.274,-55.262,172.637,21.197,153.834
C04416=1072.841,-126.522,-55.254,172.635,21.196,153.834
C04417=1072.835,-126.772,-55.244,172.634,21.195,153.834
C04418=1072.829,-127.023,-55.235,172.632,21.194,153.834
C04419=1072.823,-127.273,-55.226,172.630,21.193,153.834
C04420=1072.816,-127.522,-55.217,172.628,21.192,153.834
C04421=1072.810,-127.772,-55.208,172.627,21.192,153.834
C04422=1072.805,-128.023,-55.198,172.626,21.191,153.834
C04423=1072.801,-128.274,-55.188,172.624,21.189,153.834
C04424=1072.800,-128.525,-55.177,172.623,21.187,153.834
C04425=1072.801,-128.778,-55.165,172.622,21.183,153.834
C04426=1072.803,-129.031,-55.153,172.622,21.180,153.833
C04427=1072.809,-129.283,-55.139,172.621,21.175,153.832
C04428=1072.816,-129.534,-55.124,172.621,21.169,153.831
C04429=1072.423,-129.555,-55.284,172.575,21.304,153.863
C04430=1072.416,-129.305,-55.298,172.575,21.309,153.864
C04431=1072.411,-129.053,-55.313,172.576,21.314,153.865
C04432=1072.407,-128.800,-55.325,172.576,21.318,153.865
C04433=1072.407,-128.547,-55.338,172.577,21.321,153.866
C04434=1072.409,-128.297,-55.349,172.578,21.324,153.866
C04435=1072.412,-128.046,-55.359,172.580,21.326,153.866
C04436=1072.417,-127.795,-55.368,172.581,21.327,153.866
C04437=1072.423,-127.544,-55.377,172.583,21.327,153.866
C04438=1072.430,-127.295,-55.386,172.584,21.328,153.866
C04439=1072.435,-127.045,-55.395,172.586,21.329,153.866
C04440=1072.442,-126.795,-55.405,172.588,21.330,153.866
C04441=1072.448,-126.545,-55.414,172.589,21.330,153.866
C04442=1072.455,-126.296,-55.423,172.591,21.331,153.865
C04443=1072.461,-126.045,-55.432,172.593,21.332,153.865
C04444=1072.466,-125.796,-55.441,172.595,21.333,153.865
C04445=1072.473,-125.547,-55.450,172.596,21.334,153.865
C04446=1072.479,-125.296,-55.459,172.597,21.335,153.865
C04447=1072.485,-125.047,-55.468,172.599,21.336,153.865
C04448=1072.491,-124.797,-55.478,172.601,21.337,153.865
C04449=1072.498,-124.547,-55.487,172.602,21.337,153.865
C04450=1072.503,-124.298,-55.496,172.604,21.338,153.865
C04451=1072.510,-124.048,-55.505,172.606,21.339,153.865
C04452=1072.516,-123.798,-55.515,172.608,21.340,153.864
C04453=1072.522,-123.548,-55.524,172.609,21.341,153.864
C04454=1072.528,-123.298,-55.533,172.610,21.341,153.864
C04455=1072.534,-123.049,-55.542,172.612,21.342,153.864
C04456=1072.540,-122.799,-55.551,172.614,21.343,153.864
C04457=1072.546,-122.549,-55.561,172.615,21.344,153.864
C04458=1072.553,-122.300,-55.570,172.617,21.345,153.864
C04459=1072.559,-122.049,-55.579,172.619,21.346,153.864
C04460=1072.565,-121.799,-55.589,172.621,21.347,153.864
C04461=1072.571,-121.551,-55.597,172.622,21.348,153.864
C04462=1072.577,-121.301,-55.607,172.624,21.349,153.864
C04463=1072.583,-121.051,-55.617,172.625,21.350,153.864
C04464=1072.590,-120.801,-55.626,172.627,21.350,153.863
C04465=1072.595,-120.551,-55.635,172.628,21.351,153.863
C04466=1072.602,-120.301,-55.645,172.630,21.352,153.863
C04467=1072.608,-120.051,-55.654,172.632,21.353,153.863
C04468=1072.613,-119.802,-55.663,172.633,21.354,153.863
C04469=1072.620,-119.553,-55.672,172.635,21.355,153.863
C04470=1072.626,-119.303,-55.682,172.637,21.356,153.863
C04471=1072.633,-119.053,-55.691,172.639,21.357,153.863
C04472=1072.639,-118.803,-55.701,172.640,21.358,153.863
C04473=1072.645,-118.553,-55.710,172.641,21.359,153.863
C04474=1072.651,-118.303,-55.719,172.643,21.360,153.863
C04475=1072.657,-118.053,-55.729,172.645,21.361,153.863
C04476=1072.663,-117.804,-55.738,172.646,21.362,153.862
C04477=1072.669,-117.554,-55.748,172.648,21.363,153.862
C04478=1072.675,-117.304,-55.757,172.650,21.364,153.862
C04479=1072.681,-117.055,-55.767,172.651,21.365,153.862
C04480=1072.687,-116.805,-55.776,172.653,21.366,153.862
C04481=1072.694,-116.555,-55.785,172.655,21.367,153.862
C04482=1072.700,-116.306,-55.795,172.656,21.368,153.862
C04483=1072.706,-116.056,-55.805,172.657,21.368,153.862
C04484=1072.713,-115.806,-55.814,172.659,21.369,153.862
C04485=1072.719,-115.556,-55.824,172.661,21.371,153.862
C04486=1072.725,-115.306,-55.833,172.662,21.372,153.862
C04487=1072.731,-115.057,-55.842,172.664,21.372,153.862
C04488=1072.737,-114.807,-55.852,172.666,21.374,153.862
C04489=1072.743,-114.558,-55.862,172.668,21.375,153.862
C04490=1072.750,-114.278,-55.873,172.669,21.376,153.862
C04491=1072.756,-114.000,-55.883,172.671,21.377,153.861
C04492=1072.764,-113.721,-55.894,172.673,21.378,153.861
C04493=1072.770,-113.442,-55.905,172.674,21.379,153.861
C04494=1072.776,-113.192,-55.914,172.676,21.380,153.861
C04495=1072.782,-112.942,-55.924,172.678,21.381,153.861
C04496=1072.788,-112.693,-55.933,172.679,21.382,153.861
C04497=1072.794,-112.443,-55.943,172.681,21.384,153.861
C04498=1072.801,-112.193,-55.952,172.683,21.385,153.861
C04499=1072.807,-111.943,-55.962,172.684,21.386,153.861
C04500=1072.813,-111.693,-55.972,172.686,21.387,153.861
C04501=1072.819,-111.444,-55.981,172.687,21.388,153.861
C04502=1072.825,-111.194,-55.991,172.689,21.389,153.861
C04503=1072.831,-110.944,-56.002,172.691,21.390,153.861
C04504=1072.837,-110.694,-56.011,172.693,21.391,153.861
C04505=1072.843,-110.445,-56.021,172.694,21.393,153.861
C04506=1072.850,-110.195,-56.030,172.696,21.394,153.861
C04507=1072.856,-109.945,-56.040,172.697,21.395,153.861
C04508=1072.862,-109.695,-56.049,172.698,21.395,153.861
C04509=1072.868,-109.446,-56.059,172.700,21.397,153.861
C04510=1072.875,-109.196,-56.069,172.702,21.398,153.860
C04511=1072.881,-108.947,-56.079,172.703,21.399,153.860
C04512=1072.887,-108.697,-56.088,172.705,21.400,153.860
C04513=1072.893,-108.447,-56.098,172.707,21.401,153.860
C04514=1072.899,-108.197,-56.108,172.708,21.402,153.860
C04515=1072.905,-107.947,-56.118,172.710,21.404,153.860
C04516=1072.911,-107.698,-56.128,172.712,21.404,153.860
C04517=1072.917,-107.448,-56.138,172.713,21.406,153.860
C04518=1072.924,-107.198,-56.147,172.715,21.407,153.860
C04519=1072.930,-106.948,-56.157,172.717,21.408,153.860
C04520=1072.935,-106.698,-56.167,172.718,21.409,153.860
C04521=1072.942,-106.449,-56.177,172.720,21.410,153.860
C04522=1072.948,-106.199,-56.187,172.721,21.411,153.860
C04523=1072.954,-105.950,-56.196,172.722,21.413,153.860
C04524=1072.960,-105.700,-56.206,172.724,21.414,153.860
C04525=1072.966,-105.450,-56.217,172.725,21.415,153.860
C04526=1072.972,-105.200,-56.226,172.727,21.416,153.860
C04527=1072.978,-104.951,-56.236,172.729,21.417,153.860
C04528=1072.984,-104.701,-56.245,172.730,21.419,153.860
C04529=1072.990,-104.451,-56.256,172.732,21.420,153.860
C04530=1072.996,-104.202,-56.266,172.734,21.421,153.860
C04531=1073.002,-103.952,-56.275,172.735,21.422,153.860
C04532=1073.008,-103.702,-56.286,172.737,21.424,153.860
C04533=1073.014,-103.453,-56.296,172.738,21.425,153.860
C04534=1073.021,-103.203,-56.305,172.740,21.426,153.860
C04535=1073.027,-102.954,-56.316,172.742,21.427,153.860
C04536=1073.032,-102.703,-56.326,172.743,21.429,153.860
C04537=1073.039,-102.454,-56.335,172.745,21.430,153.860
C04538=1073.045,-102.204,-56.346,172.746,21.431,153.860
C04539=1073.051,-101.954,-56.356,172.748,21.432,153.860
C04540=1073.057,-101.704,-56.366,172.750,21.434,153.860
C04541=1073.064,-101.455,-56.376,172.751,21.435,153.860
C04542=1073.070,-101.205,-56.386,172.753,21.436,153.860
C04543=1073.075,-100.955,-56.396,172.754,21.437,153.860
C04544=1073.082,-100.706,-56.406,172.755,21.438,153.860
C04545=1073.088,-100.456,-56.416,172.757,21.439,153.860
C04546=1073.094,-100.206,-56.427,172.759,21.441,153.860
C04547=1073.100,-99.957,-56.436,172.760,21.442,153.860
C04548=1073.106,-99.707,-56.446,172.762,21.444,153.860
C04549=1073.112,-99.457,-56.457,172.763,21.445,153.860
C04550=1073.119,-99.207,-56.467,172.765,21.446,153.860
C04551=1073.125,-98.958,-56.477,172.767,21.447,153.860
C04552=1073.131,-98.707,-56.487,172.768,21.449,153.860
C04553=1073.137,-98.458,-56.497,172.770,21.450,153.860
C04554=1073.144,-98.176,-56.509,172.771,21.451,153.860
C04555=1073.151,-97.895,-56.520,172.774,21.453,153.860
C04556=1073.157,-97.614,-56.532,172.775,21.455,153.860
C04557=1073.164,-97.332,-56.542,172.777,21.456,153.860
C04558=1073.171,-97.082,-56.553,172.778,21.457,153.860
C04559=1073.177,-96.832,-56.563,172.780,21.459,153.860
C04560=1073.182,-96.583,-56.574,172.782,21.460,153.859
C04561=1073.189,-96.333,-56.583,172.783,21.461,153.860
C04562=1073.194,-96.084,-56.594,172.785,21.462,153.860
C04563=1073.201,-95.834,-56.604,172.786,21.464,153.860
C04564=1073.206,-95.584,-56.615,172.788,21.465,153.860
C04565=1073.212,-95.334,-56.625,172.789,21.467,153.860
C04566=1073.218,-95.085,-56.635,172.791,21.468,153.860
C04567=1073.224,-94.836,-56.646,172.793,21.469,153.860
C04568=1073.231,-94.585,-56.656,172.794,21.471,153.860
C04569=1073.236,-94.336,-56.667,172.796,21.472,153.860
C04570=1073.243,-94.086,-56.676,172.797,21.474,153.860
C04571=1073.248,-93.836,-56.687,172.799,21.475,153.860
C04572=1073.255,-93.587,-56.697,172.800,21.477,153.860
C04573=1073.260,-93.337,-56.708,172.802,21.478,153.860
C04574=1073.266,-93.088,-56.718,172.804,21.479,153.860
C04575=1073.273,-92.837,-56.728,172.805,21.481,153.860
C04576=1073.279,-92.588,-56.739,172.807,21.482,153.860
C04577=1073.285,-92.338,-56.749,172.808,21.484,153.860
C04578=1073.290,-92.088,-56.760,172.810,21.485,153.860
C04579=1073.297,-91.839,-56.770,172.811,21.487,153.860
C04580=1073.302,-91.589,-56.780,172.813,21.488,153.860
C04581=1073.309,-91.339,-56.791,172.814,21.490,153.860
C04582=1073.315,-91.090,-56.802,172.816,21.491,153.860
C04583=1073.321,-90.840,-56.812,172.817,21.492,153.860
C04584=1073.327,-90.590,-56.822,172.819,21.494,153.860
C04585=1073.333,-90.341,-56.833,172.820,21.495,153.860
C04586=1073.339,-90.091,-56.843,172.822,21.497,153.860
C04587=1073.345,-89.841,-56.854,172.824,21.498,153.860
C04588=1073.351,-89.591,-56.865,172.825,21.499,153.860
C04589=1073.357,-89.342,-56.874,172.827,21.501,153.860
C04590=1073.363,-89.092,-56.885,172.828,21.502,153.860
C04591=1073.370,-88.842,-56.896,172.830,21.504,153.860
C04592=1073.375,-88.592,-56.906,172.831,21.506,153.860
C04593=1073.381,-88.343,-56.917,172.833,21.507,153.860
C04594=1073.388,-88.093,-56.927,172.834,21.508,153.860
C04595=1073.393,-87.844,-56.938,172.836,21.510,153.860
C04596=1073.399,-87.593,-56.949,172.837,21.511,153.860
C04597=1073.406,-87.344,-56.959,172.839,21.513,153.860
C04598=1073.412,-87.094,-56.970,172.841,21.514,153.860
C04599=1073.418,-86.845,-56.980,172.842,21.516,153.861
C04600=1073.424,-86.594,-56.991,172.844,21.517,153.861
C04601=1073.430,-86.345,-57.001,172.845,21.519,153.861
C04602=1073.436,-86.096,-57.012,172.847,21.520,153.861
C04603=1073.442,-85.846,-57.023,172.848,21.522,153.861
C04604=1073.448,-85.596,-57.034,172.850,21.523,153.861
C04605=1073.455,-85.346,-57.043,172.851,21.525,153.861
C04606=1073.460,-85.097,-57.054,172.853,21.526,153.861
C04607=1073.467,-84.847,-57.065,172.854,21.528,153.861
C04608=1073.473,-84.597,-57.076,172.856,21.529,153.861
C04609=1073.479,-84.348,-57.087,172.857,21.531,153.861
C04610=1073.485,-84.098,-57.096,172.859,21.533,153.861
C04611=1073.491,-83.848,-57.107,172.860,21.534,153.861
C04612=1073.497,-83.598,-57.118,172.862,21.535,153.861
C04613=1073.504,-83.349,-57.129,172.863,21.537,153.861
C04614=1073.510,-83.099,-57.140,172.865,21.538,153.861
C04615=1073.516,-82.850,-57.151,172.866,21.540,153.861
C04616=1073.522,-82.600,-57.161,172.868,21.541,153.861
C04617=1073.529,-82.350,-57.172,172.870,21.543,153.861
C04618=1073.535,-82.071,-57.184,172.871,21.544,153.861
C04619=1073.542,-81.792,-57.196,172.872,21.546,153.862
C04620=1073.548,-81.513,-57.208,172.874,21.548,153.862
C04621=1073.556,-81.233,-57.220,172.876,21.550,153.862
C04622=1073.562,-80.984,-57.231,172.878,21.551,153.862
C04623=1073.568,-80.735,-57.242,172.879,21.553,153.862
C04624=1073.575,-80.485,-57.253,172.881,21.554,153.862
C04625=1073.580,-80.235,-57.264,172.882,21.556,153.862
C04626=1073.586,-79.985,-57.274,172.884,21.558,153.862
C04627=1073.593,-79.735,-57.284,172.885,21.559,153.862
C04628=1073.599,-79.486,-57.295,172.887,21.561,153.862
C04629=1073.604,-79.236,-57.306,172.888,21.562,153.862
C04630=1073.611,-78.986,-57.317,172.890,21.564,153.862
C04631=1073.616,-78.736,-57.328,172.891,21.566,153.862
C04632=1073.622,-78.487,-57.339,172.893,21.567,153.862
C04633=1073.628,-78.237,-57.350,172.894,21.568,153.862
C04634=1073.635,-77.988,-57.361,172.896,21.570,153.862
C04635=1073.641,-77.738,-57.372,172.897,21.572,153.862
C04636=1073.647,-77.488,-57.383,172.899,21.574,153.863
C04637=1073.653,-77.238,-57.394,172.900,21.575,153.863
C04638=1073.659,-76.989,-57.405,172.902,21.577,153.863
C04639=1073.665,-76.739,-57.417,172.903,21.578,153.863
C04640=1073.671,-76.490,-57.427,172.905,21.580,153.863
C04641=1073.677,-76.240,-57.439,172.906,21.582,153.863
C04642=1073.683,-75.990,-57.450,172.908,21.583,153.863
C04643=1073.689,-75.741,-57.460,172.909,21.585,153.863
C04644=1073.696,-75.491,-57.471,172.911,21.587,153.863
C04645=1073.701,-75.241,-57.482,172.912,21.588,153.863
C04646=1073.707,-74.992,-57.493,172.914,21.590,153.863
C04647=1073.714,-74.742,-57.504,172.915,21.592,153.863
C04648=1073.719,-74.492,-57.515,172.917,21.594,153.863
C04649=1073.726,-74.242,-57.526,172.919,21.595,153.863
C04650=1073.732,-73.993,-57.538,172.920,21.597,153.864
C04651=1073.737,-73.744,-57.549,172.922,21.599,153.864
C04652=1073.744,-73.493,-57.560,172.923,21.600,153.864
C04653=1073.750,-73.244,-57.571,172.925,21.602,153.864
C04654=1073.755,-72.994,-57.582,172.926,21.604,153.864
C04655=1073.761,-72.744,-57.594,172.928,21.606,153.864
C04656=1073.767,-72.494,-57.604,172.929,21.608,153.864
C04657=1073.773,-72.245,-57.616,172.930,21.609,153.864
C04658=1073.779,-71.995,-57.627,172.932,21.611,153.864
C04659=1073.785,-71.746,-57.638,172.933,21.612,153.864
C04660=1073.791,-71.496,-57.649,172.935,21.614,153.865
C04661=1073.797,-71.246,-57.660,172.936,21.616,153.865
C04662=1073.802,-70.997,-57.672,172.938,21.618,153.865
C04663=1073.808,-70.747,-57.684,172.939,21.620,153.865
C04664=1073.814,-70.497,-57.695,172.940,21.622,153.865
C04665=1073.821,-70.247,-57.706,172.942,21.623,153.865
C04666=1073.826,-69.998,-57.717,172.943,21.625,153.865
C04667=1073.832,-69.749,-57.728,172.945,21.626,153.865
C04668=1073.839,-69.499,-57.739,172.946,21.628,153.865
C04669=1073.844,-69.249,-57.751,172.948,21.630,153.866
C04670=1073.850,-68.999,-57.763,172.950,21.632,153.866
C04671=1073.856,-68.750,-57.774,172.951,21.634,153.866
C04672=1073.862,-68.500,-57.785,172.953,21.636,153.866
C04673=1073.868,-68.250,-57.796,172.954,21.637,153.866
C04674=1073.874,-68.001,-57.808,172.956,21.639,153.866
C04675=1073.880,-67.751,-57.819,172.957,21.641,153.866
C04676=1073.886,-67.501,-57.830,172.959,21.643,153.866
C04677=1073.892,-67.252,-57.842,172.960,21.644,153.866
C04678=1073.898,-67.002,-57.853,172.961,21.646,153.867
C04679=1073.904,-66.752,-57.864,172.963,21.648,153.867
C04680=1073.910,-66.503,-57.876,172.964,21.650,153.867
C04681=1073.916,-66.252,-57.888,172.966,21.652,153.867
C04682=1073.922,-65.976,-57.900,172.967,21.654,153.867
C04683=1073.929,-65.699,-57.913,172.969,21.656,153.867
C04684=1073.936,-65.422,-57.926,172.971,21.658,153.867
C04685=1073.943,-65.145,-57.938,172.972,21.660,153.867
C04686=1073.949,-64.896,-57.950,172.974,21.661,153.867
C04687=1073.954,-64.645,-57.961,172.975,21.663,153.868
C04688=1073.960,-64.396,-57.972,172.976,21.665,153.868
C04689=1073.967,-64.146,-57.984,172.979,21.667,153.868
C04690=1073.972,-63.897,-57.995,172.980,21.669,153.868
C04691=1073.979,-63.647,-58.007,172.982,21.671,153.868
C04692=1073.984,-63.397,-58.019,172.983,21.673,153.868
C04693=1073.990,-63.147,-58.030,172.985,21.674,153.868
C04694=1073.996,-62.898,-58.041,172.986,21.676,153.868
C04695=1074.003,-62.648,-58.053,172.987,21.678,153.869
C04696=1074.008,-62.399,-58.065,172.989,21.680,153.869
C04697=1074.014,-62.149,-58.076,172.990,21.682,153.869
C04698=1074.020,-61.900,-58.088,172.992,21.683,153.869
C04699=1074.027,-61.650,-58.099,172.993,21.685,153.869
C04700=1074.032,-61.400,-58.111,172.994,21.687,153.869
C04701=1074.038,-61.150,-58.122,172.996,21.689,153.869
C04702=1074.045,-60.901,-58.134,172.997,21.691,153.869
C04703=1074.051,-60.651,-58.145,172.999,21.693,153.870
C04704=1074.057,-60.401,-58.158,173.001,21.695,153.870
C04705=1074.062,-60.152,-58.169,173.002,21.697,153.870
C04706=1074.069,-59.902,-58.181,173.004,21.699,153.870
C04707=1074.075,-59.653,-58.191,173.005,21.700,153.870
C04708=1074.081,-59.403,-58.204,173.007,21.702,153.870
C04709=1074.087,-59.153,-58.215,173.008,21.704,153.870
C04710=1074.093,-58.904,-58.227,173.009,21.706,153.870
C04711=1074.099,-58.654,-58.239,173.011,21.708,153.871
C04712=1074.105,-58.404,-58.250,173.012,21.709,153.871
C04713=1074.111,-58.155,-58.262,173.014,21.711,153.871
C04714=1074.118,-57.905,-58.274,173.015,21.713,153.871
C04715=1074.123,-57.655,-58.286,173.016,21.715,153.871
C04716=1074.129,-57.405,-58.297,173.018,21.717,153.871
C04717=1074.136,-57.156,-58.309,173.019,21.719,153.871
C04718=1074.141,-56.907,-58.321,173.022,21.721,153.871
C04719=1074.148,-56.656,-58.332,173.023,21.723,153.871
C04720=1074.154,-56.407,-58.344,173.024,21.725,153.872
C04721=1074.160,-56.158,-58.356,173.026,21.727,153.872
C04722=1074.166,-55.907,-58.368,173.027,21.729,153.872
C04723=1074.172,-55.659,-58.379,173.028,21.731,153.872
C04724=1074.179,-55.409,-58.391,173.030,21.732,153.872
C04725=1074.184,-55.158,-58.403,173.031,21.734,153.872
C04726=1074.190,-54.910,-58.415,173.033,21.736,153.872
C04727=1074.197,-54.660,-58.427,173.034,21.738,153.873
C04728=1074.203,-54.409,-58.439,173.035,21.740,153.873
C04729=1074.209,-54.161,-58.450,173.037,21.742,153.873
C04730=1074.215,-53.911,-58.462,173.039,21.744,153.873
C04731=1074.221,-53.661,-58.474,173.040,21.746,153.873
C04732=1074.228,-53.411,-58.486,173.042,21.747,153.873
C04733=1074.234,-53.162,-58.497,173.043,21.749,153.873
C04734=1074.239,-52.912,-58.510,173.045,21.751,153.873
C04735=1074.246,-52.662,-58.521,173.046,21.753,153.874
C04736=1074.252,-52.413,-58.533,173.048,21.755,153.874
C04737=1074.258,-52.163,-58.545,173.049,21.757,153.874
C04738=1074.264,-51.914,-58.557,173.050,21.759,153.874
C04739=1074.270,-51.663,-58.569,173.052,21.761,153.874
C04740=1074.276,-51.414,-58.581,173.053,21.763,153.874
C04741=1074.283,-51.165,-58.593,173.054,21.765,153.875
C04742=1074.289,-50.915,-58.605,173.057,21.767,153.875
C04743=1074.294,-50.665,-58.616,173.058,21.769,153.875
C04744=1074.301,-50.416,-58.628,173.060,21.771,153.875
C04745=1074.307,-50.166,-58.641,173.061,21.772,153.875
C04746=1074.314,-49.891,-58.654,173.062,21.775,153.875
C04747=1074.320,-49.615,-58.667,173.064,21.777,153.875
C04748=1074.327,-49.339,-58.681,173.066,21.779,153.876
C04749=1074.333,-49.063,-58.694,173.067,21.781,153.876
C04750=1074.339,-48.813,-58.706,173.068,21.784,153.876
C04751=1074.345,-48.564,-58.718,173.070,21.786,153.876
C04752=1074.351,-48.315,-58.730,173.071,21.788,153.876
C04753=1074.357,-48.065,-58.743,173.072,21.790,153.876
C04754=1074.362,-47.816,-58.755,173.075,21.792,153.877
C04755=1074.369,-47.566,-58.767,173.076,21.794,153.877
C04756=1074.375,-47.315,-58.779,173.077,21.796,153.877
C04757=1074.381,-47.066,-58.791,173.079,21.798,153.877
C04758=1074.387,-46.817,-58.803,173.080,21.800,153.877
C04759=1074.393,-46.567,-58.815,173.082,21.802,153.877
C04760=1074.398,-46.317,-58.828,173.083,21.804,153.878
C04761=1074.404,-46.068,-58.840,173.084,21.806,153.878
C04762=1074.410,-45.818,-58.852,173.086,21.808,153.878
C04763=1074.416,-45.568,-58.865,173.087,21.810,153.878
C04764=1074.423,-45.319,-58.877,173.088,21.812,153.878
C04765=1074.428,-45.070,-58.889,173.091,21.814,153.878
C04766=1074.434,-44.820,-58.901,173.092,21.816,153.879
C04767=1074.441,-44.570,-58.913,173.093,21.818,153.879
C04768=1074.447,-44.320,-58.926,173.094,21.820,153.879
C04769=1074.452,-44.071,-58.938,173.096,21.822,153.879
C04770=1074.459,-43.821,-58.950,173.097,21.824,153.879
C04771=1074.465,-43.572,-58.963,173.099,21.826,153.879
C04772=1074.470,-43.322,-58.975,173.100,21.828,153.880
C04773=1074.477,-43.073,-58.987,173.101,21.830,153.880
C04774=1074.482,-42.823,-58.999,173.103,21.832,153.880
C04775=1074.488,-42.573,-59.012,173.105,21.835,153.880
C04776=1074.495,-42.324,-59.024,173.106,21.837,153.880
C04777=1074.501,-42.074,-59.036,173.108,21.839,153.880
C04778=1074.506,-41.824,-59.049,173.109,21.841,153.881
C04779=1074.512,-41.575,-59.061,173.110,21.843,153.881
C04780=1074.519,-41.325,-59.073,173.112,21.845,153.881
C04781=1074.525,-41.075,-59.086,173.113,21.847,153.881
C04782=1074.531,-40.825,-59.098,173.114,21.849,153.881
C04783=1074.536,-40.575,-59.111,173.116,21.851,153.882
C04784=1074.543,-40.326,-59.122,173.118,21.853,153.882
C04785=1074.548,-40.077,-59.135,173.119,21.855,153.882
C04786=1074.555,-39.827,-59.148,173.120,21.858,153.882
C04787=1074.561,-39.578,-59.160,173.122,21.860,153.882
C04788=1074.567,-39.328,-59.173,173.123,21.862,153.882
C04789=1074.573,-39.078,-59.185,173.125,21.864,153.883
C04790=1074.578,-38.829,-59.197,173.126,21.866,153.883
C04791=1074.585,-38.579,-59.209,173.127,21.867,153.883
C04792=1074.591,-38.329,-59.222,173.129,21.870,153.883
C04793=1074.597,-38.080,-59.235,173.131,21.872,153.883
C04794=1074.603,-37.830,-59.248,173.132,21.874,153.883
C04795=1074.609,-37.580,-59.260,173.133,21.877,153.884
C04796=1074.614,-37.331,-59.272,173.135,21.879,153.884
C04797=1074.620,-37.081,-59.285,173.136,21.881,153.884
C04798=1074.626,-36.831,-59.298,173.137,21.883,153.884
C04799=1074.632,-36.582,-59.311,173.139,21.885,153.884
C04800=1074.638,-36.332,-59.323,173.140,21.887,153.885
C04801=1074.644,-36.082,-59.336,173.141,21.889,153.885
C04802=1074.649,-35.833,-59.348,173.143,21.892,153.885
C04803=1074.656,-35.584,-59.361,173.145,21.894,153.885
C04804=1074.662,-35.334,-59.373,173.146,21.896,153.885
C04805=1074.668,-35.084,-59.386,173.147,21.898,153.886
C04806=1074.674,-34.835,-59.398,173.149,21.900,153.886
C04807=1074.680,-34.585,-59.412,173.150,21.902,153.886
C04808=1074.686,-34.335,-59.424,173.151,21.904,153.886
C04809=1074.692,-34.086,-59.436,173.153,21.906,153.886
C04810=1074.698,-33.811,-59.451,173.155,21.909,153.887
C04811=1074.705,-33.536,-59.465,173.156,21.911,153.887
C04812=1074.711,-33.261,-59.478,173.157,21.914,153.887
C04813=1074.717,-32.985,-59.493,173.160,21.916,153.887
C04814=1074.724,-32.736,-59.506,173.161,21.919,153.887
C04815=1074.730,-32.486,-59.518,173.162,21.920,153.888
C04816=1074.736,-32.236,-59.531,173.164,21.922,153.888
C04817=1074.742,-31.987,-59.544,173.165,21.925,153.888
C04818=1074.748,-31.737,-59.557,173.166,21.927,153.888
C04819=1074.754,-31.487,-59.569,173.167,21.929,153.888
C04820=1074.760,-31.238,-59.583,173.170,21.932,153.889
C04821=1074.766,-30.988,-59.595,173.171,21.934,153.889
C04822=1074.772,-30.738,-59.608,173.172,21.936,153.889
C04823=1074.778,-30.488,-59.621,173.174,21.938,153.889
C04824=1074.784,-30.239,-59.634,173.175,21.940,153.889
C04825=1074.790,-29.989,-59.647,173.176,21.942,153.890
C04826=1074.795,-29.740,-59.659,173.178,21.944,153.890
C04827=1074.801,-29.491,-59.672,173.179,21.946,153.890
C04828=1074.807,-29.241,-59.685,173.181,21.949,153.890
C04829=1074.813,-28.991,-59.697,173.182,21.951,153.890
C04830=1074.819,-28.742,-59.711,173.184,21.954,153.891
C04831=1074.825,-28.492,-59.723,173.185,21.955,153.891
C04832=1074.832,-28.243,-59.736,173.186,21.957,153.891
C04833=1074.837,-27.993,-59.749,173.188,21.960,153.891
C04834=1074.844,-27.744,-59.762,173.189,21.962,153.891
C04835=1074.850,-27.494,-59.775,173.190,21.964,153.892
C04836=1074.856,-27.244,-59.788,173.192,21.967,153.892
C04837=1074.862,-26.995,-59.801,173.194,21.969,153.892
C04838=1074.868,-26.745,-59.814,173.195,21.971,153.892
C04839=1074.874,-26.495,-59.826,173.196,21.973,153.892
C04840=1074.880,-26.246,-59.840,173.198,21.975,153.893
C04841=1074.886,-25.996,-59.852,173.199,21.977,153.893
C04842=1074.891,-25.747,-59.866,173.200,21.980,153.893
C04843=1074.897,-25.497,-59.879,173.201,21.982,153.893
C04844=1074.904,-25.248,-59.892,173.204,21.985,153.894
C04845=1074.909,-24.998,-59.905,173.205,21.987,153.894
C04846=1074.915,-24.748,-59.918,173.206,21.989,153.894
C04847=1074.921,-24.498,-59.931,173.208,21.991,153.894
C04848=1074.927,-24.249,-59.944,173.209,21.993,153.894
C04849=1074.933,-23.999,-59.957,173.210,21.995,153.895
C04850=1074.939,-23.750,-59.970,173.211,21.998,153.895
C04851=1074.945,-23.500,-59.984,173.213,22.000,153.895
C04852=1074.951,-23.250,-59.996,173.215,22.003,153.895
C04853=1074.957,-23.001,-60.010,173.216,22.005,153.895
C04854=1074.963,-22.752,-60.023,173.217,22.007,153.896
C04855=1074.968,-22.502,-60.036,173.219,22.009,153.896
C04856=1074.974,-22.252,-60.049,173.220,22.011,153.896
C04857=1074.980,-22.002,-60.062,173.221,22.013,153.896
C04858=1074.987,-21.753,-60.075,173.223,22.016,153.897
C04859=1074.992,-21.504,-60.089,173.225,22.018,153.897
C04860=1074.998,-21.254,-60.102,173.226,22.021,153.897
C04861=1075.004,-21.004,-60.115,173.227,22.023,153.897
C04862=1075.010,-20.755,-60.128,173.229,22.025,153.897
C04863=1075.016,-20.505,-60.141,173.230,22.027,153.898
C04864=1075.022,-20.256,-60.155,173.231,22.029,153.898
C04865=1075.028,-20.006,-60.168,173.233,22.031,153.898
C04866=1075.033,-19.756,-60.181,173.234,22.034,153.898
C04867=1075.040,-19.506,-60.195,173.236,22.037,153.899
C04868=1075.046,-19.257,-60.208,173.237,22.039,153.899
C04869=1075.052,-19.008,-60.221,173.238,22.041,153.899
C04870=1075.058,-18.758,-60.234,173.240,22.043,153.899
C04871=1075.064,-18.508,-60.248,173.241,22.045,153.899
C04872=1075.070,-18.259,-60.261,173.242,22.047,153.900
C04873=1075.075,-18.009,-60.275,173.244,22.050,153.900
C04874=1075.082,-17.733,-60.289,173.246,22.053,153.900
C04875=1075.089,-17.457,-60.304,173.247,22.055,153.900
C04876=1075.096,-17.181,-60.319,173.248,22.057,153.901
C04877=1075.102,-16.905,-60.334,173.250,22.060,153.901
C04878=1075.108,-16.655,-60.347,173.251,22.063,153.901
C04879=1075.115,-16.406,-60.360,173.253,22.064,153.901
C04880=1075.120,-16.156,-60.373,173.254,22.067,153.902
C04881=1075.126,-15.907,-60.387,173.255,22.069,153.902
C04882=1075.132,-15.657,-60.400,173.258,22.072,153.902
C04883=1075.138,-15.408,-60.414,173.259,22.074,153.902
C04884=1075.145,-15.158,-60.427,173.260,22.076,153.902
C04885=1075.151,-14.909,-60.441,173.262,22.078,153.903
C04886=1075.156,-14.658,-60.454,173.263,22.080,153.903
C04887=1075.162,-14.409,-60.467,173.264,22.083,153.903
C04888=1075.168,-14.160,-60.481,173.265,22.085,153.903
C04889=1075.174,-13.910,-60.494,173.267,22.088,153.904
C04890=1075.179,-13.661,-60.508,173.269,22.090,153.904
C04891=1075.186,-13.411,-60.521,173.270,22.092,153.904
C04892=1075.191,-13.162,-60.535,173.271,22.095,153.904
C04893=1075.197,-12.912,-60.549,173.272,22.097,153.905
C04894=1075.203,-12.662,-60.563,173.274,22.099,153.905
C04895=1075.209,-12.413,-60.576,173.275,22.101,153.905
C04896=1075.215,-12.163,-60.589,173.277,22.104,153.905
C04897=1075.220,-11.913,-60.603,173.278,22.106,153.905
C04898=1075.226,-11.664,-60.616,173.280,22.109,153.906
C04899=1075.232,-11.414,-60.630,173.281,22.111,153.906
C04900=1075.239,-11.164,-60.644,173.282,22.113,153.906
C04901=1075.244,-10.915,-60.658,173.283,22.116,153.907
C04902=1075.250,-10.666,-60.671,173.285,22.118,153.907
C04903=1075.256,-10.416,-60.685,173.287,22.120,153.907
C04904=1075.262,-10.167,-60.698,173.288,22.123,153.907
C04905=1075.268,-9.917,-60.712,173.289,22.125,153.907
C04906=1075.274,-9.667,-60.725,173.291,22.127,153.908
C04907=1075.280,-9.418,-60.739,173.292,22.130,153.908
C04908=1075.285,-9.168,-60.753,173.293,22.132,153.908
C04909=1075.291,-8.919,-60.766,173.295,22.134,153.908
C04910=1075.297,-8.669,-60.780,173.297,22.137,153.909
C04911=1075.304,-8.419,-60.794,173.298,22.139,153.909
C04912=1075.309,-8.170,-60.808,173.299,22.141,153.909
C04913=1075.315,-7.920,-60.821,173.300,22.144,153.909
C04914=1075.321,-7.672,-60.836,173.302,22.146,153.910
C04915=1075.327,-7.422,-60.849,173.303,22.148,153.910
C04916=1075.334,-7.172,-60.863,173.304,22.151,153.910
C04917=1075.339,-6.922,-60.877,173.306,22.154,153.910
C04918=1075.345,-6.673,-60.890,173.308,22.155,153.911
C04919=1075.351,-6.424,-60.904,173.309,22.158,153.911
C04920=1075.358,-6.174,-60.918,173.310,22.160,153.911
C04921=1075.363,-5.924,-60.932,173.311,22.163,153.911
C04922=1075.368,-5.674,-60.945,173.313,22.165,153.912
C04923=1075.375,-5.426,-60.959,173.315,22.168,153.912
C04924=1075.381,-5.176,-60.974,173.316,22.170,153.912
C04925=1075.387,-4.926,-60.987,173.317,22.172,153.912
C04926=1075.393,-4.677,-61.001,173.319,22.174,153.913
C04927=1075.399,-4.426,-61.015,173.320,22.177,153.913
C04928=1075.405,-4.177,-61.028,173.321,22.179,153.913
C04929=1075.411,-3.928,-61.042,173.322,22.181,153.913
C04930=1075.416,-3.679,-61.057,173.324,22.184,153.914
C04931=1075.423,-3.429,-61.070,173.326,22.186,153.914
C04932=1075.429,-3.179,-61.084,173.327,22.189,153.914
C04933=1075.434,-2.929,-61.098,173.328,22.191,153.914
C04934=1075.440,-2.681,-61.113,173.329,22.193,153.915
C04935=1075.447,-2.431,-61.126,173.331,22.196,153.915
C04936=1075.452,-2.181,-61.140,173.333,22.198,153.915
C04937=1075.458,-1.931,-61.154,173.334,22.201,153.915
C04938=1075.464,-1.654,-61.170,173.335,22.203,153.916
C04939=1075.470,-1.376,-61.186,173.337,22.206,153.916
C04940=1075.477,-1.098,-61.201,173.339,22.209,153.916
C04941=1075.483,-0.821,-61.217,173.340,22.212,153.916
C04942=1075.489,-0.571,-61.231,173.341,22.214,153.917
C04943=1075.495,-0.321,-61.245,173.343,22.216,153.917
C04944=1075.501,-0.072,-61.260,173.344,22.219,153.917
C04945=1075.507,0.177,-61.273,173.346,22.221,153.917
C04946=1075.513,0.428,-61.287,173.347,22.224,153.918
C04947=1075.519,0.677,-61.302,173.348,22.226,153.918
C04948=1075.524,0.926,-61.316,173.349,22.228,153.918
C04949=1075.530,1.176,-61.329,173.352,22.231,153.918
C04950=1075.536,1.425,-61.344,173.353,22.233,153.919
C04951=1075.542,1.675,-61.358,173.354,22.236,153.919
C04952=1075.547,1.924,-61.372,173.355,22.238,153.919
C04953=1075.553,2.174,-61.387,173.356,22.241,153.920
C04954=1075.560,2.423,-61.400,173.358,22.243,153.920
C04955=1075.565,2.672,-61.415,173.360,22.246,153.920
C04956=1075.572,2.923,-61.429,173.361,22.248,153.920
C04957=1075.577,3.172,-61.443,173.362,22.250,153.921
C04958=1075.583,3.421,-61.458,173.363,22.253,153.921
C04959=1075.589,3.671,-61.472,173.365,22.255,153.921
C04960=1075.595,3.920,-61.486,173.366,22.257,153.921
C04961=1075.600,4.170,-61.500,173.368,22.260,153.922
C04962=1075.606,4.420,-61.514,173.369,22.263,153.922
C04963=1075.612,4.669,-61.529,173.371,22.265,153.922
C04964=1075.618,4.919,-61.543,173.372,22.268,153.922
C04965=1075.624,5.168,-61.558,173.373,22.269,153.923
C04966=1075.630,5.418,-61.571,173.374,22.272,153.923
C04967=1075.636,5.667,-61.586,173.376,22.274,153.923
C04968=1075.642,5.917,-61.600,173.378,22.277,153.923
C04969=1075.648,6.166,-61.615,173.379,22.280,153.924
C04970=1075.654,6.416,-61.629,173.380,22.282,153.924
C04971=1075.660,6.665,-61.643,173.382,22.284,153.924
C04972=1075.665,6.915,-61.657,173.383,22.286,153.925
C04973=1075.671,7.164,-61.672,173.384,22.289,153.925
C04974=1075.677,7.414,-61.686,173.386,22.292,153.925
C04975=1075.683,7.664,-61.701,173.387,22.294,153.925
C04976=1075.689,7.913,-61.715,173.389,22.296,153.925
C04977=1075.695,8.162,-61.729,173.390,22.299,153.926
C04978=1075.701,8.412,-61.744,173.391,22.301,153.926
C04979=1075.706,8.661,-61.758,173.392,22.304,153.926
C04980=1075.713,8.911,-61.773,173.394,22.306,153.927
C04981=1075.718,9.161,-61.787,173.396,22.308,153.927
C04982=1075.725,9.410,-61.802,173.397,22.311,153.927
C04983=1075.730,9.660,-61.816,173.398,22.313,153.927
C04984=1075.737,9.909,-61.831,173.400,22.316,153.928
C04985=1075.742,10.158,-61.845,173.401,22.318,153.928
C04986=1075.748,10.408,-61.859,173.403,22.321,153.928
C04987=1075.754,10.658,-61.874,173.404,22.323,153.928
C04988=1075.760,10.907,-61.888,173.405,22.325,153.929
C04989=1075.766,11.157,-61.903,173.407,22.328,153.929
C04990=1075.772,11.406,-61.918,173.408,22.330,153.929
C04991=1075.778,11.656,-61.932,173.409,22.333,153.930
C04992=1075.784,11.905,-61.946,173.411,22.335,153.930
C04993=1075.790,12.155,-61.961,173.413,22.337,153.930
C04994=1075.796,12.404,-61.975,173.414,22.340,153.930
C04995=1075.802,12.654,-61.990,173.415,22.342,153.931
C04996=1075.808,12.903,-62.005,173.416,22.345,153.931
C04997=1075.814,13.153,-62.020,173.419,22.347,153.931
C04998=1075.820,13.402,-62.034,173.420,22.350,153.931
C04999=1075.826,13.652,-62.048,173.421,22.352,153.931
C05000=1075.832,13.901,-62.063,173.422,22.355,153.932
C05001=1075.838,14.151,-62.077,173.423,22.357,153.932
C05002=1075.845,14.430,-62.094,173.426,22.360,153.932
C05003=1075.851,14.710,-62.110,173.427,22.362,153.933
C05004=1075.857,14.990,-62.127,173.429,22.365,153.933
C05005=1075.864,15.269,-62.144,173.430,22.368,153.933
C05006=1075.870,15.519,-62.158,173.431,22.370,153.933
C05007=1075.876,15.768,-62.172,173.433,22.372,153.934
C05008=1075.882,16.018,-62.188,173.434,22.375,153.934
C05009=1075.888,16.267,-62.203,173.436,22.378,153.934
C05010=1075.894,16.517,-62.218,173.437,22.380,153.935
C05011=1075.899,16.767,-62.231,173.438,22.383,153.935
C05012=1075.905,17.017,-62.247,173.439,22.385,153.935
C05013=1075.911,17.266,-62.262,173.441,22.388,153.935
C05014=1075.917,17.515,-62.276,173.443,22.390,153.936
C05015=1075.923,17.764,-62.291,173.444,22.393,153.936
C05016=1075.929,18.014,-62.307,173.445,22.395,153.936
C05017=1075.934,18.263,-62.321,173.447,22.397,153.936
C05018=1075.940,18.513,-62.335,173.448,22.400,153.937
C05019=1075.946,18.762,-62.350,173.449,22.402,153.937
C05020=1075.952,19.012,-62.366,173.451,22.405,153.937
C05021=1075.958,19.261,-62.380,173.452,22.407,153.938
C05022=1075.964,19.511,-62.395,173.454,22.410,153.938
C05023=1075.970,19.761,-62.410,173.455,22.412,153.938
C05024=1075.975,20.010,-62.425,173.456,22.415,153.938
C05025=1075.982,20.259,-62.440,173.458,22.417,153.939
C05026=1075.988,20.508,-62.455,173.460,22.420,153.939
C05027=1075.993,20.758,-62.470,173.461,22.422,153.939
C05028=1075.999,21.007,-62.485,173.462,22.424,153.939
C05029=1076.005,21.258,-62.499,173.463,22.427,153.940
C05030=1076.011,21.508,-62.515,173.465,22.429,153.940
C05031=1076.017,21.757,-62.529,173.467,22.432,153.940
C05032=1076.023,22.006,-62.544,173.468,22.435,153.941
C05033=1076.028,22.255,-62.559,173.469,22.437,153.941
C05034=1076.034,22.505,-62.574,173.470,22.440,153.941
C05035=1076.039,22.754,-62.589,173.472,22.442,153.941
C05036=1076.046,23.004,-62.604,173.474,22.445,153.942
C05037=1076.052,23.254,-62.619,173.475,22.447,153.942
C05038=1076.057,23.503,-62.634,173.476,22.450,153.942
C05039=1076.064,23.753,-62.649,173.477,22.452,153.943
C05040=1076.069,24.001,-62.665,173.479,22.454,153.943
C05041=1076.075,24.251,-62.680,173.481,22.457,153.943
C05042=1076.082,24.501,-62.695,173.482,22.459,153.943
C05043=1076.087,24.750,-62.710,173.483,22.462,153.944
C05044=1076.093,24.999,-62.725,173.485,22.464,153.944
C05045=1076.098,25.249,-62.740,173.486,22.467,153.944
C05046=1076.105,25.498,-62.755,173.487,22.469,153.944
C05047=1076.111,25.748,-62.770,173.489,22.472,153.945
C05048=1076.116,25.997,-62.786,173.490,22.474,153.945
C05049=1076.122,26.247,-62.801,173.492,22.477,153.945
C05050=1076.128,26.497,-62.816,173.493,22.479,153.946
C05051=1076.134,26.746,-62.831,173.494,22.481,153.946
C05052=1076.140,26.995,-62.847,173.496,22.484,153.946
C05053=1076.146,27.245,-62.862,173.498,22.486,153.946
C05054=1076.151,27.494,-62.877,173.499,22.489,153.947
C05055=1076.158,27.744,-62.892,173.500,22.491,153.947
C05056=1076.164,27.993,-62.907,173.501,22.494,153.947
C05057=1076.169,28.243,-62.922,173.503,22.497,153.947
C05058=1076.176,28.492,-62.938,173.505,22.499,153.948
C05059=1076.181,28.742,-62.953,173.506,22.502,153.948
C05060=1076.187,28.991,-62.968,173.507,22.504,153.948
C05061=1076.193,29.241,-62.983,173.508,22.506,153.949
C05062=1076.198,29.491,-62.999,173.510,22.509,153.949
C05063=1076.205,29.739,-63.014,173.512,22.512,153.949
C05064=1076.210,29.989,-63.030,173.513,22.514,153.949
C05065=1076.217,30.239,-63.045,173.514,22.517,153.950
C05066=1076.222,30.520,-63.062,173.516,22.519,153.950
C05067=1076.229,30.801,-63.079,173.517,22.522,153.950
C05068=1076.236,31.082,-63.097,173.519,22.525,153.951
C05069=1076.242,31.363,-63.114,173.521,22.528,153.951
C05070=1076.248,31.612,-63.130,173.522,22.530,153.951
C05071=1076.253,31.861,-63.145,173.524,22.533,153.951
C05072=1076.260,32.111,-63.160,173.525,22.535,153.952
C05073=1076.265,32.361,-63.176,173.526,22.538,153.952
C05074=1076.271,32.609,-63.191,173.528,22.540,153.952
C05075=1076.277,32.859,-63.207,173.529,22.543,153.953
C05076=1076.283,33.109,-63.222,173.531,22.546,153.953
C05077=1076.289,33.358,-63.238,173.532,22.548,153.953
C05078=1076.295,33.608,-63.253,173.533,22.550,153.953
C05079=1076.300,33.858,-63.269,173.535,22.553,153.954
C05080=1076.307,34.107,-63.284,173.536,22.555,153.954
C05081=1076.312,34.356,-63.299,173.538,22.558,153.954
C05082=1076.318,34.605,-63.316,173.539,22.561,153.955
C05083=1076.324,34.855,-63.331,173.540,22.563,153.955
C05084=1076.330,35.105,-63.346,173.542,22.565,153.955
C05085=1076.335,35.354,-63.362,173.543,22.567,153.955
C05086=1076.342,35.603,-63.377,173.545,22.570,153.956
C05087=1076.348,35.853,-63.393,173.546,22.573,153.956
C05088=1076.353,36.103,-63.409,173.548,22.575,153.956
C05089=1076.360,36.352,-63.424,173.549,22.578,153.956
C05090=1076.365,36.601,-63.440,173.550,22.580,153.957
C05091=1076.371,36.851,-63.455,173.552,22.583,153.957
C05092=1076.377,37.100,-63.471,173.554,22.585,153.957
C05093=1076.383,37.350,-63.486,173.555,22.588,153.958
C05094=1076.388,37.598,-63.502,173.556,22.590,153.958
C05095=1076.394,37.848,-63.518,173.558,22.593,153.958
C05096=1076.401,38.097,-63.533,173.559,22.595,153.958
C05097=1076.406,38.347,-63.549,173.561,22.598,153.959
C05098=1076.412,38.597,-63.565,173.562,22.600,153.959
C05099=1076.417,38.846,-63.580,173.563,22.603,153.959
C05100=1076.423,39.095,-63.597,173.565,22.606,153.960
C05101=1076.429,39.345,-63.612,173.566,22.608,153.960
C05102=1076.436,39.594,-63.628,173.568,22.610,153.960
C05103=1076.441,39.844,-63.643,173.569,22.613,153.960
C05104=1076.447,40.093,-63.659,173.570,22.615,153.961
C05105=1076.452,40.343,-63.675,173.572,22.618,153.961
C05106=1076.458,40.592,-63.691,173.573,22.621,153.961
C05107=1076.464,40.842,-63.707,173.575,22.623,153.962
C05108=1076.469,41.091,-63.723,173.576,22.625,153.962
C05109=1076.476,41.340,-63.738,173.578,22.628,153.962
C05110=1076.481,41.590,-63.754,173.579,22.631,153.962
C05111=1076.487,41.839,-63.770,173.581,22.633,153.963
C05112=1076.493,42.089,-63.786,173.582,22.636,153.963
C05113=1076.498,42.338,-63.801,173.583,22.638,153.963
C05114=1076.504,42.587,-63.818,173.585,22.641,153.964
C05115=1076.510,42.837,-63.833,173.587,22.643,153.964
C05116=1076.516,43.087,-63.849,173.588,22.645,153.964
C05117=1076.522,43.336,-63.866,173.589,22.648,153.964
C05118=1076.528,43.586,-63.881,173.591,22.650,153.965
C05119=1076.534,43.835,-63.897,173.592,22.653,153.965
C05120=1076.539,44.084,-63.913,173.594,22.655,153.965
C05121=1076.544,44.334,-63.929,173.595,22.658,153.965
C05122=1076.550,44.583,-63.945,173.596,22.661,153.966
C05123=1076.556,44.833,-63.961,173.598,22.664,153.966
C05124=1076.562,45.083,-63.977,173.599,22.666,153.966
C05125=1076.567,45.331,-63.993,173.601,22.668,153.967
C05126=1076.573,45.581,-64.009,173.602,22.671,153.967
C05127=1076.579,45.830,-64.025,173.604,22.674,153.967
C05128=1076.585,46.080,-64.041,173.605,22.676,153.968
C05129=1076.591,46.329,-64.057,173.606,22.679,153.968
C05130=1076.597,46.610,-64.076,173.609,22.681,153.968
C05131=1076.603,46.891,-64.094,173.610,22.684,153.968
C05132=1076.609,47.172,-64.112,173.612,22.687,153.969
C05133=1076.616,47.453,-64.129,173.613,22.690,153.969
C05134=1076.622,47.703,-64.146,173.614,22.693,153.969
C05135=1076.628,47.952,-64.162,173.616,22.695,153.970
C05136=1076.634,48.202,-64.179,173.617,22.698,153.970
C05137=1076.639,48.450,-64.195,173.619,22.700,153.970
C05138=1076.645,48.700,-64.211,173.620,22.703,153.971
C05139=1076.650,48.950,-64.226,173.622,22.706,153.971
C05140=1076.656,49.199,-64.243,173.623,22.708,153.971
C05141=1076.662,49.448,-64.259,173.625,22.710,153.971
C05142=1076.668,49.698,-64.276,173.626,22.713,153.972
C05143=1076.674,49.948,-64.292,173.627,22.715,153.972
C05144=1076.680,50.197,-64.308,173.629,22.718,153.972
C05145=1076.685,50.446,-64.325,173.630,22.720,153.973
C05146=1076.691,50.696,-64.340,173.632,22.723,153.973
C05147=1076.696,50.945,-64.356,173.633,22.725,153.973
C05148=1076.702,51.194,-64.373,173.635,22.728,153.973
C05149=1076.708,51.444,-64.389,173.636,22.731,153.974
C05150=1076.714,51.693,-64.405,173.638,22.733,153.974
C05151=1076.720,51.943,-64.422,173.639,22.735,153.974
C05152=1076.725,52.192,-64.438,173.641,22.738,153.975
C05153=1076.731,52.441,-64.454,173.642,22.741,153.975
C05154=1076.737,52.691,-64.471,173.643,22.743,153.975
C05155=1076.743,52.940,-64.487,173.645,22.746,153.975
C05156=1076.749,53.190,-64.503,173.647,22.748,153.976
C05157=1076.754,53.439,-64.520,173.648,22.751,153.976
C05158=1076.760,53.688,-64.536,173.649,22.753,153.976
C05159=1076.766,53.938,-64.552,173.651,22.756,153.977
C05160=1076.772,54.187,-64.569,173.653,22.758,153.977
C05161=1076.778,54.437,-64.585,173.654,22.760,153.977
C05162=1076.784,54.686,-64.602,173.655,22.763,153.977
C05163=1076.789,54.935,-64.618,173.657,22.765,153.978
C05164=1076.795,55.185,-64.634,173.659,22.768,153.978
C05165=1076.801,55.434,-64.651,173.660,22.770,153.978
C05166=1076.807,55.684,-64.667,173.661,22.773,153.978
C05167=1076.813,55.933,-64.683,173.662,22.775,153.979
C05168=1076.818,56.182,-64.700,173.665,22.778,153.979
C05169=1076.824,56.432,-64.716,173.666,22.781,153.979
C05170=1076.830,56.681,-64.733,173.667,22.783,153.980
C05171=1076.836,56.931,-64.749,173.668,22.785,153.980
C05172=1076.842,57.180,-64.765,173.671,22.788,153.980
C05173=1076.847,57.429,-64.782,173.672,22.791,153.980
C05174=1076.853,57.678,-64.799,173.673,22.793,153.981
C05175=1076.859,57.928,-64.815,173.674,22.796,153.981
C05176=1076.865,58.177,-64.832,173.677,22.798,153.981
C05177=1076.871,58.427,-64.848,173.678,22.800,153.981
C05178=1076.876,58.676,-64.865,173.679,22.803,153.982
C05179=1076.882,58.926,-64.881,173.680,22.805,153.982
C05180=1076.889,59.176,-64.898,173.682,22.808,153.982
C05181=1076.895,59.424,-64.915,173.684,22.810,153.982
C05182=1076.900,59.674,-64.931,173.685,22.813,153.983
C05183=1076.906,59.923,-64.948,173.686,22.815,153.983
C05184=1076.912,60.173,-64.964,173.688,22.818,153.983
C05185=1076.918,60.422,-64.980,173.690,22.820,153.984
C05186=1076.923,60.671,-64.998,173.691,22.822,153.984
C05187=1076.929,60.920,-65.014,173.693,22.825,153.984
C05188=1076.935,61.170,-65.030,173.694,22.828,153.984
C05189=1076.941,61.420,-65.048,173.696,22.830,153.985
C05190=1076.947,61.669,-65.065,173.697,22.832,153.985
C05191=1076.953,61.918,-65.081,173.699,22.835,153.985
C05192=1076.959,62.168,-65.097,173.700,22.838,153.985
C05193=1076.965,62.417,-65.114,173.702,22.840,153.986
C05194=1076.971,62.698,-65.133,173.704,22.843,153.986
C05195=1076.978,62.979,-65.152,173.705,22.845,153.986
C05196=1076.984,63.259,-65.170,173.707,22.848,153.987
C05197=1076.992,63.540,-65.189,173.708,22.851,153.987
C05198=1076.997,63.789,-65.206,173.711,22.853,153.987
C05199=1077.004,64.039,-65.223,173.712,22.856,153.987
C05200=1077.010,64.289,-65.239,173.713,22.858,153.988
C05201=1077.015,64.538,-65.257,173.714,22.861,153.988
C05202=1077.021,64.787,-65.273,173.716,22.863,153.988
C05203=1077.026,65.037,-65.290,173.718,22.866,153.989
C05204=1077.033,65.286,-65.307,173.719,22.868,153.989
C05205=1077.038,65.535,-65.323,173.720,22.871,153.989
C05206=1077.045,65.785,-65.341,173.723,22.873,153.989
C05207=1077.050,66.034,-65.358,173.724,22.875,153.990
C05208=1077.056,66.284,-65.374,173.725,22.878,153.990
C05209=1077.061,66.533,-65.392,173.727,22.881,153.990
C05210=1077.067,66.782,-65.408,173.728,22.883,153.990
C05211=1077.073,67.031,-65.425,173.730,22.885,153.991
C05212=1077.079,67.280,-65.442,173.731,22.888,153.991
C05213=1077.085,67.531,-65.459,173.733,22.891,153.991
C05214=1077.091,67.780,-65.476,173.734,22.893,153.992
C05215=1077.096,68.029,-65.493,173.736,22.895,153.992
C05216=1077.102,68.278,-65.510,173.738,22.898,153.992
C05217=1077.107,68.528,-65.526,173.739,22.901,153.992
C05218=1077.113,68.777,-65.544,173.740,22.903,153.993
C05219=1077.120,69.027,-65.561,173.742,22.905,153.993
C05220=1077.125,69.276,-65.578,173.744,22.908,153.993
C05221=1077.131,69.525,-65.594,173.745,22.910,153.993
C05222=1077.137,69.774,-65.612,173.746,22.913,153.994
C05223=1077.142,70.024,-65.629,173.749,22.915,153.994
C05224=1077.149,70.273,-65.646,173.750,22.918,153.994
C05225=1077.154,70.523,-65.663,173.751,22.920,153.995
C05226=1077.159,70.772,-65.681,173.752,22.923,153.995
C05227=1077.165,71.021,-65.697,173.754,22.926,153.995
C05228=1077.171,71.270,-65.714,173.756,22.928,153.995
C05229=1077.176,71.519,-65.732,173.757,22.930,153.996
C05230=1077.183,71.769,-65.749,173.759,22.933,153.996
C05231=1077.188,72.018,-65.766,173.760,22.936,153.996
C05232=1077.194,72.268,-65.783,173.762,22.937,153.996
C05233=1077.200,72.517,-65.800,173.763,22.940,153.997
C05234=1077.206,72.767,-65.818,173.765,22.943,153.997
C05235=1077.211,73.016,-65.835,173.767,22.945,153.997
C05236=1077.217,73.265,-65.852,173.768,22.948,153.998
C05237=1077.223,73.515,-65.869,173.770,22.950,153.998
C05238=1077.228,73.764,-65.886,173.771,22.953,153.998
C05239=1077.234,74.013,-65.904,173.772,22.955,153.998
C05240=1077.240,74.263,-65.921,173.775,22.958,153.999
C05241=1077.246,74.512,-65.938,173.776,22.960,153.999
C05242=1077.251,74.761,-65.956,173.777,22.963,153.999
C05243=1077.257,75.011,-65.973,173.779,22.965,153.999
C05244=1077.263,75.260,-65.990,173.781,22.967,154.000
C05245=1077.269,75.509,-66.007,173.782,22.970,154.000
C05246=1077.274,75.758,-66.025,173.783,22.972,154.000
C05247=1077.280,76.008,-66.042,173.785,22.975,154.000
C05248=1077.286,76.257,-66.060,173.787,22.978,154.001
C05249=1077.292,76.506,-66.077,173.788,22.980,154.001
C05250=1077.298,76.756,-66.095,173.790,22.983,154.001
C05251=1077.303,77.005,-66.111,173.792,22.985,154.001
C05252=1077.309,77.255,-66.129,173.793,22.987,154.002
C05253=1077.316,77.504,-66.146,173.794,22.989,154.002
C05254=1077.321,77.753,-66.164,173.796,22.992,154.002
C05255=1077.326,78.003,-66.181,173.798,22.995,154.003
C05256=1077.332,78.252,-66.198,173.799,22.997,154.003
C05257=1077.338,78.501,-66.216,173.801,23.000,154.003
C05258=1077.345,78.782,-66.236,173.802,23.002,154.003
C05259=1077.351,79.063,-66.256,173.804,23.005,154.004
C05260=1077.357,79.343,-66.275,173.807,23.008,154.004
C05261=1077.364,79.624,-66.295,173.808,23.011,154.004
C05262=1077.370,79.874,-66.312,173.809,23.013,154.005
C05263=1077.375,80.123,-66.330,173.811,23.016,154.005
C05264=1077.381,80.372,-66.347,173.812,23.018,154.005
C05265=1077.387,80.622,-66.365,173.814,23.020,154.005
C05266=1077.392,80.871,-66.383,173.816,23.023,154.006
C05267=1077.398,81.120,-66.400,173.817,23.026,154.006
C05268=1077.403,81.369,-66.418,173.818,23.028,154.006
C05269=1077.410,81.619,-66.436,173.821,23.031,154.007
C05270=1077.415,81.868,-66.453,173.822,23.033,154.007
C05271=1077.420,82.117,-66.470,173.823,23.036,154.007
C05272=1077.426,82.367,-66.488,173.825,23.038,154.007
C05273=1077.432,82.616,-66.506,173.827,23.041,154.008
C05274=1077.437,82.865,-66.523,173.828,23.043,154.008
C05275=1077.444,83.115,-66.541,173.830,23.045,154.008
C05276=1077.449,83.364,-66.559,173.831,23.048,154.008
C05277=1077.455,83.613,-66.576,173.833,23.050,154.009
C05278=1077.461,83.863,-66.594,173.835,23.053,154.009
C05279=1077.466,84.112,-66.612,173.836,23.055,154.009
C05280=1077.472,84.362,-66.630,173.837,23.058,154.010
C05281=1077.478,84.611,-66.647,173.840,23.060,154.010
C05282=1077.483,84.860,-66.665,173.841,23.063,154.010
C05283=1077.489,85.109,-66.683,173.842,23.065,154.010
C05284=1077.495,85.358,-66.700,173.844,23.068,154.010
C05285=1077.501,85.607,-66.718,173.846,23.070,154.011
C05286=1077.507,85.857,-66.736,173.847,23.073,154.011
C05287=1077.512,86.106,-66.753,173.849,23.075,154.011
C05288=1077.518,86.356,-66.771,173.851,23.077,154.012
C05289=1077.523,86.605,-66.790,173.852,23.080,154.012
C05290=1077.530,86.854,-66.808,173.854,23.082,154.012
C05291=1077.535,87.103,-66.826,173.855,23.085,154.012
C05292=1077.541,87.353,-66.843,173.857,23.087,154.013
C05293=1077.547,87.602,-66.861,173.859,23.090,154.013
C05294=1077.552,87.851,-66.879,173.860,23.092,154.013
C05295=1077.558,88.101,-66.897,173.861,23.094,154.013
C05296=1077.564,88.350,-66.914,173.864,23.097,154.014
C05297=1077.570,88.599,-66.933,173.865,23.100,154.014
C05298=1077.576,88.848,-66.951,173.866,23.101,154.014
C05299=1077.582,89.098,-66.968,173.869,23.104,154.014
C05300=1077.587,89.347,-66.986,173.870,23.107,154.015
C05301=1077.594,89.597,-67.004,173.871,23.109,154.015
C05302=1077.599,89.846,-67.022,173.873,23.111,154.015
C05303=1077.604,90.095,-67.040,173.875,23.114,154.015
C05304=1077.610,90.344,-67.058,173.876,23.116,154.016
C05305=1077.616,90.593,-67.076,173.878,23.119,154.016
C05306=1077.622,90.843,-67.094,173.880,23.121,154.016
C05307=1077.627,91.092,-67.111,173.881,23.123,154.016
C05308=1077.634,91.341,-67.130,173.883,23.126,154.017
C05309=1077.639,91.591,-67.148,173.884,23.128,154.017
C05310=1077.645,91.840,-67.166,173.886,23.131,154.017
C05311=1077.650,92.089,-67.184,173.888,23.134,154.017
C05312=1077.657,92.338,-67.202,173.889,23.136,154.018
C05313=1077.661,92.588,-67.221,173.891,23.138,154.018
C05314=1077.668,92.838,-67.238,173.893,23.141,154.018
C05315=1077.673,93.086,-67.257,173.894,23.143,154.019
C05316=1077.679,93.336,-67.275,173.896,23.146,154.019
C05317=1077.684,93.585,-67.293,173.897,23.148,154.019
C05318=1077.691,93.834,-67.311,173.899,23.150,154.019
C05319=1077.696,94.084,-67.330,173.901,23.153,154.019
C05320=1077.702,94.333,-67.348,173.902,23.155,154.020
C05321=1077.707,94.582,-67.366,173.904,23.158,154.020
C05322=1077.714,94.863,-67.386,173.906,23.160,154.020
C05323=1077.719,95.144,-67.407,173.908,23.163,154.021
C05324=1077.726,95.425,-67.428,173.909,23.166,154.021
C05325=1077.733,95.706,-67.448,173.911,23.168,154.021
C05326=1077.738,95.954,-67.466,173.913,23.171,154.021
C05327=1077.744,96.204,-67.484,173.915,23.174,154.022
C05328=1077.750,96.453,-67.503,173.916,23.176,154.022
C05329=1077.756,96.702,-67.521,173.918,23.179,154.022
C05330=1077.762,96.951,-67.539,173.920,23.181,154.022
C05331=1077.767,97.201,-67.557,173.921,23.183,154.023
C05332=1077.773,97.451,-67.575,173.923,23.186,154.023
C05333=1077.778,97.699,-67.594,173.924,23.188,154.023
C05334=1077.784,97.949,-67.612,173.927,23.190,154.023
C05335=1077.790,98.197,-67.631,173.928,23.193,154.024
C05336=1077.795,98.447,-67.649,173.929,23.195,154.024
C05337=1077.802,98.697,-67.668,173.931,23.198,154.024
C05338=1077.807,98.946,-67.685,173.933,23.200,154.024
C05339=1077.813,99.195,-67.705,173.934,23.202,154.025
C05340=1077.819,99.444,-67.722,173.936,23.205,154.025
C05341=1077.824,99.694,-67.741,173.938,23.207,154.025
C05342=1077.830,99.943,-67.759,173.940,23.210,154.025
C05343=1077.836,100.192,-67.778,173.941,23.212,154.026
C05344=1077.842,100.441,-67.797,173.943,23.215,154.026
C05345=1077.847,100.690,-67.814,173.945,23.217,154.026
C05346=1077.853,100.940,-67.834,173.946,23.219,154.026
C05347=1077.859,101.189,-67.852,173.947,23.222,154.027
C05348=1077.865,101.438,-67.870,173.950,23.224,154.027
C05349=1077.870,101.688,-67.888,173.951,23.226,154.027
C05350=1077.876,101.937,-67.907,173.953,23.229,154.027
C05351=1077.882,102.186,-67.926,173.955,23.231,154.028
C05352=1077.887,102.436,-67.944,173.956,23.234,154.028
C05353=1077.893,102.684,-67.963,173.958,23.236,154.028
C05354=1077.899,102.934,-67.982,173.959,23.238,154.028
C05355=1077.904,103.183,-68.000,173.962,23.241,154.029
C05356=1077.910,103.432,-68.019,173.963,23.244,154.029
C05357=1077.916,103.681,-68.038,173.964,23.246,154.029
C05358=1077.921,103.930,-68.056,173.967,23.248,154.029
C05359=1077.927,104.180,-68.075,173.968,23.251,154.030
C05360=1077.933,104.429,-68.094,173.970,23.253,154.030
C05361=1077.938,104.678,-68.112,173.972,23.255,154.030
C05362=1077.944,104.928,-68.131,173.973,23.258,154.030
C05363=1077.950,105.176,-68.149,173.975,23.261,154.031
C05364=1077.955,105.426,-68.168,173.976,23.263,154.031
C05365=1077.961,105.676,-68.187,173.979,23.265,154.031
C05366=1077.967,105.924,-68.205,173.980,23.268,154.031
C05367=1077.972,106.174,-68.224,173.981,23.270,154.032
C05368=1077.978,106.424,-68.243,173.984,23.272,154.032
C05369=1077.983,106.672,-68.261,173.985,23.275,154.032
C05370=1077.989,106.922,-68.280,173.987,23.277,154.032
C05371=1077.996,107.171,-68.299,173.988,23.280,154.033
C05372=1078.001,107.419,-68.318,173.991,23.282,154.033
C05373=1078.006,107.669,-68.337,173.992,23.284,154.033
C05374=1078.012,107.919,-68.355,173.993,23.287,154.033
C05375=1078.018,108.168,-68.374,173.996,23.289,154.034
C05376=1078.023,108.417,-68.393,173.997,23.291,154.034
C05377=1078.030,108.666,-68.412,173.999,23.294,154.034
C05378=1078.035,108.915,-68.431,174.000,23.296,154.034
C05379=1078.040,109.164,-68.450,174.002,23.298,154.035
C05380=1078.047,109.414,-68.468,174.004,23.301,154.035
C05381=1078.052,109.663,-68.487,174.005,23.303,154.035
C05382=1078.058,109.913,-68.506,174.008,23.306,154.035
C05383=1078.064,110.161,-68.525,174.009,23.308,154.036
C05384=1078.069,110.410,-68.544,174.011,23.311,154.036
C05385=1078.075,110.660,-68.563,174.013,23.313,154.036
C05386=1078.082,110.941,-68.584,174.015,23.316,154.036
C05387=1078.088,111.221,-68.606,174.016,23.318,154.037
C05388=1078.094,111.503,-68.627,174.018,23.321,154.037
C05389=1078.101,111.783,-68.648,174.020,23.324,154.037
C05390=1078.107,112.032,-68.667,174.022,23.325,154.037
C05391=1078.112,112.282,-68.687,174.024,23.328,154.037
C05392=1078.118,112.531,-68.706,174.025,23.331,154.038
C05393=1078.124,112.780,-68.724,174.028,23.333,154.038
C05394=1078.130,113.029,-68.743,174.029,23.335,154.038
C05395=1078.135,113.279,-68.763,174.031,23.338,154.038
C05396=1078.141,113.528,-68.782,174.033,23.340,154.039
C05397=1078.146,113.777,-68.801,174.034,23.342,154.039
C05398=1078.152,114.026,-68.820,174.036,23.345,154.039
C05399=1078.158,114.275,-68.839,174.038,23.347,154.039
C05400=1078.164,114.525,-68.858,174.040,23.350,154.040
C05401=1078.170,114.774,-68.877,174.041,23.352,154.040
C05402=1078.178,115.175,-68.908,174.044,23.356,154.040
C05403=1078.187,115.577,-68.940,174.047,23.360,154.041
C05404=1078.196,115.978,-68.970,174.050,23.364,154.041
C05405=1078.205,116.380,-69.002,174.053,23.367,154.041
C05406=1078.211,116.630,-69.021,174.055,23.370,154.042
C05407=1078.216,116.879,-69.040,174.056,23.373,154.042
C05408=1078.221,117.128,-69.059,174.057,23.374,154.042
C05409=1078.227,117.377,-69.078,174.060,23.377,154.042
C05410=1078.233,117.627,-69.097,174.061,23.380,154.043
C05411=1078.239,117.876,-69.117,174.063,23.382,154.043
C05412=1078.244,118.125,-69.137,174.065,23.384,154.043
C05413=1078.249,118.374,-69.155,174.067,23.387,154.043
C05414=1078.255,118.623,-69.175,174.068,23.389,154.044
C05415=1078.261,118.873,-69.194,174.070,23.392,154.044
C05416=1078.267,119.121,-69.214,174.072,23.394,154.044
C05417=1078.273,119.371,-69.233,174.074,23.396,154.044
C05418=1078.277,119.620,-69.253,174.075,23.399,154.045
C05419=1078.283,119.869,-69.272,174.078,23.401,154.045
C05420=1078.289,120.118,-69.292,174.079,23.403,154.045
C05421=1078.294,120.368,-69.311,174.080,23.406,154.045
C05422=1078.300,120.617,-69.330,174.083,23.408,154.045
C05423=1078.306,120.866,-69.350,174.084,23.410,154.046
C05424=1078.312,121.115,-69.370,174.086,23.413,154.046
C05425=1078.317,121.364,-69.388,174.088,23.415,154.046
C05426=1078.322,121.613,-69.408,174.090,23.418,154.046
C05427=1078.328,121.862,-69.428,174.091,23.420,154.047
C05428=1078.334,122.112,-69.447,174.094,23.422,154.047
C05429=1078.340,122.361,-69.466,174.095,23.425,154.047
C05430=1078.345,122.610,-69.487,174.097,23.427,154.047
C05431=1078.351,122.860,-69.506,174.099,23.429,154.048
C05432=1078.356,123.109,-69.525,174.101,23.432,154.048
C05433=1078.362,123.358,-69.545,174.102,23.434,154.048
C05434=1078.367,123.607,-69.564,174.104,23.437,154.048
C05435=1078.373,123.855,-69.584,174.106,23.439,154.048
C05436=1078.379,124.105,-69.603,174.108,23.441,154.049
C05437=1078.385,124.354,-69.622,174.109,23.444,154.049
C05438=1078.390,124.603,-69.643,174.112,23.446,154.049
C05439=1078.396,124.853,-69.662,174.113,23.448,154.049
C05440=1078.402,125.102,-69.682,174.115,23.451,154.049
C05441=1078.407,125.351,-69.701,174.117,23.453,154.050
C05442=1078.413,125.600,-69.721,174.119,23.455,154.050
C05443=1078.419,125.849,-69.741,174.120,23.458,154.050
C05444=1078.425,126.098,-69.761,174.123,23.460,154.050
C05445=1078.430,126.348,-69.780,174.124,23.462,154.051
C05446=1078.439,126.725,-69.810,174.127,23.466,154.051
C05447=1078.447,127.103,-69.840,174.130,23.470,154.051
C05448=1078.456,127.480,-69.869,174.133,23.473,154.052
C05449=1078.465,127.857,-69.900,174.135,23.476,154.052
C05450=1078.471,128.107,-69.919,174.137,23.479,154.052
C05451=1078.477,128.356,-69.939,174.139,23.481,154.052
C05452=1078.482,128.605,-69.958,174.141,23.483,154.053
C05453=1078.488,128.854,-69.978,174.142,23.485,154.053
C05454=1078.493,129.104,-69.998,174.145,23.488,154.053
C05455=1078.499,129.352,-70.018,174.146,23.490,154.053
C05456=1078.505,129.601,-70.038,174.148,23.492,154.053
C05457=1078.511,129.851,-70.057,174.150,23.494,154.054
C05458=1078.517,130.100,-70.077,174.152,23.497,154.054
